LIN {X 0,Y 464.494,Z 1183.228,A -85,B 0,C 180,E1 15563.324,E2 15563.324} C_VEL
LIN {X 0,Y 465.219,Z 1176.701,A -85,B 0,C 180,E1 15560.224,E2 15560.224} C_VEL
LIN {X 0,Y 466.194,Z 1170.108,A -85,B 0,C 180,E1 15557.615,E2 15557.615} C_VEL
LIN {X 0,Y 467.574,Z 1162.416,A -85,B 0,C 180,E1 15555.004,E2 15555.004} C_VEL
LIN {X 0,Y 469.489,Z 1153.124,A -85,B 0,C 180,E1 15552.269,E2 15552.269} C_VEL
LIN {X 0,Y 472.708,Z 1139.667,A -85,B 0,C 180,E1 15548.88,E2 15548.88} C_VEL
LIN {X 0,Y 475.924,Z 1127.311,A -85,B 0,C 180,E1 15546.21,E2 15546.21} C_VEL
LIN {X 0,Y 479.291,Z 1115.185,A -85,B 0,C 180,E1 15543.884,E2 15543.884} C_VEL
LIN {X 0,Y 482.99,Z 1102.43,A -85,B 0,C 180,E1 15541.701,E2 15541.701} C_VEL
LIN {X 0,Y 487.449,Z 1087.469,A -85,B 0,C 180,E1 15539.422,E2 15539.422} C_VEL
LIN {X 0,Y 493.552,Z 1066.908,A -85,B 0,C 180,E1 15536.7,E2 15536.7} C_VEL
LIN {X 0,Y 498.429,Z 1050.219,A -85,B 0,C 180,E1 15534.778,E2 15534.778} C_VEL
LIN {X 0,Y 503.252,Z 1033.414,A -85,B 0,C 180,E1 15533.057,E2 15533.057} C_VEL
LIN {X 0,Y 508.073,Z 1016.053,A -85,B 0,C 180,E1 15531.474,E2 15531.474} C_VEL
LIN {X 0,Y 513.784,Z 994.616,A -85,B 0,C 180,E1 15529.751,E2 15529.751} C_VEL
LIN {X 0,Y 519.62,Z 970.597,A -85,B 0,C 180,E1 15528.109,E2 15528.109} C_VEL
LIN {X 0,Y 524.036,Z 951.032,A -85,B 0,C 180,E1 15526.953,E2 15526.953} C_VEL
LIN {X 0,Y 527.937,Z 932.043,A -85,B 0,C 180,E1 15525.967,E2 15525.967} C_VEL
LIN {X 0,Y 531.669,Z 912.17,A -85,B 0,C 180,E1 15525.075,E2 15525.075} C_VEL
LIN {X 0,Y 535.289,Z 890.47,A -85,B 0,C 180,E1 15524.246,E2 15524.246} C_VEL
LIN {X 0,Y 539.188,Z 862.655,A -85,B 0,C 180,E1 15523.385,E2 15523.385} C_VEL
LIN {X 0,Y 541.832,Z 838.413,A -85,B 0,C 180,E1 15522.811,E2 15522.811} C_VEL
LIN {X 0,Y 543.64,Z 816.068,A -85,B 0,C 180,E1 15522.403,E2 15522.403} C_VEL
LIN {X 0,Y 553.541,Z 604.138,A -85,B 0,C 180,E1 15519.202,E2 15519.202} C_VEL
LIN {X 0,Y 559.827,Z 471.624,A -85,B 0,C 180,E1 15517.173,E2 15517.173} C_VEL
LIN {X 0,Y 549.211,Z 455.582,A -85,B 0,C 180,E1 15515.058,E2 15515.058} C_VEL
LIN {X 0,Y 537.64,Z 439.734,A -85,B 0,C 180,E1 15512.544,E2 15512.544} C_VEL
LIN {X 0,Y 528.377,Z 427.759,A -85,B 0,C 180,E1 15510.318,E2 15510.318} C_VEL
LIN {X 0,Y 521.179,Z 418.584,A -85,B 0,C 180,E1 15508.411,E2 15508.411} C_VEL
LIN {X 0,Y 516.1,Z 412.456,A -85,B 0,C 180,E1 15506.959,E2 15506.959} C_VEL
LIN {X 0,Y 511.821,Z 407.184,A -85,B 0,C 180,E1 15505.641,E2 15505.641} C_VEL
LIN {X 0,Y 508.019,Z 402.462,A -85,B 0,C 180,E1 15504.383,E2 15504.383} C_VEL
LIN {X 0,Y 503.556,Z 397.56,A -85,B 0,C 180,E1 15502.812,E2 15502.812} C_VEL
LIN {X 0,Y 502.199,Z 395.757,A -85,B 0,C 180,E1 15502.29,E2 15502.29} C_VEL
LIN {X 0,Y 498.68,Z 392.223,A -85,B 0,C 180,E1 15500.91,E2 15500.91} C_VEL
LIN {X 0,Y 496.917,Z 389.555,A -85,B 0,C 180,E1 15500.126,E2 15500.126} C_VEL
LIN {X 0,Y 493.635,Z 386.766,A -85,B 0,C 180,E1 15498.665,E2 15498.665} C_VEL
LIN {X 0,Y 491.477,Z 383.313,A -85,B 0,C 180,E1 15497.524,E2 15497.524} C_VEL
LIN {X 0,Y 488.072,Z 380.844,A -85,B 0,C 180,E1 15495.69,E2 15495.69} C_VEL
LIN {X 0,Y 486.117,Z 377.519,A -85,B 0,C 180,E1 15494.353,E2 15494.353} C_VEL
LIN {X 0,Y 485.736,Z 376.677,A -85,B 0,C 180,E1 15494.058,E2 15494.058} C_VEL
LIN {X 0,Y 481.79,Z 374.262,A -85,B 0,C 180,E1 15490.997,E2 15490.997} C_VEL
LIN {X 0,Y 480.013,Z 370.955,A -85,B 0,C 180,E1 15488.807,E2 15488.807} C_VEL
LIN {X 0,Y 479.704,Z 369.991,A -85,B 0,C 180,E1 15488.269,E2 15488.269} C_VEL
LIN {X 0,Y 477.971,Z 369.512,A -85,B 0,C 180,E1 15481.558,E2 15481.558} C_VEL
LIN {X 0,Y 479.808,Z 370.162,A -85,B 0,C 180,E1 15477.671,E2 15477.671} C_VEL
LIN {X 0,Y 481.494,Z 373.959,A -85,B 0,C 180,E1 15475.4,E2 15475.4} C_VEL
LIN {X 0,Y 484.978,Z 376.507,A -85,B 0,C 180,E1 15472.537,E2 15472.537} C_VEL
LIN {X 0,Y 485.888,Z 377.026,A -85,B 0,C 180,E1 15471.926,E2 15471.926} C_VEL
LIN {X 0,Y 487.83,Z 380.574,A -85,B 0,C 180,E1 15470.562,E2 15470.562} C_VEL
LIN {X 0,Y 490.711,Z 382.963,A -85,B 0,C 180,E1 15468.957,E2 15468.957} C_VEL
LIN {X 0,Y 491.78,Z 383.73,A -85,B 0,C 180,E1 15468.417,E2 15468.417} C_VEL
LIN {X 0,Y 494.132,Z 387.367,A -85,B 0,C 180,E1 15467.198,E2 15467.198} C_VEL
LIN {X 0,Y 497.51,Z 390.286,A -85,B 0,C 180,E1 15465.718,E2 15465.718} C_VEL
LIN {X 0,Y 500.44,Z 394.393,A -85,B 0,C 180,E1 15464.47,E2 15464.47} C_VEL
LIN {X 0,Y 502.915,Z 396.596,A -85,B 0,C 180,E1 15463.542,E2 15463.542} C_VEL
LIN {X 0,Y 506.304,Z 400.928,A -85,B 0,C 180,E1 15462.294,E2 15462.294} C_VEL
LIN {X 0,Y 508.201,Z 402.882,A -85,B 0,C 180,E1 15461.651,E2 15461.651} C_VEL
LIN {X 0,Y 512.093,Z 407.534,A -85,B 0,C 180,E1 15460.376,E2 15460.376} C_VEL
LIN {X 0,Y 517.261,Z 413.691,A -85,B 0,C 180,E1 15458.809,E2 15458.809} C_VEL
LIN {X 0,Y 525.953,Z 424.62,A -85,B 0,C 180,E1 15456.41,E2 15456.41} C_VEL
LIN {X 0,Y 535.695,Z 438.163,A -85,B 0,C 180,E1 15453.983,E2 15453.983} C_VEL
LIN {X 0,Y 545.364,Z 452.379,A -85,B 0,C 180,E1 15451.799,E2 15451.799} C_VEL
LIN {X 0,Y 557.011,Z 470.151,A -85,B 0,C 180,E1 15449.409,E2 15449.409} C_VEL
LIN {X 0,Y 559.909,Z 475.043,A -85,B 0,C 180,E1 15448.84,E2 15448.84} C_VEL
LIN {X 0,Y 549.743,Z 688.806,A -85,B 0,C 180,E1 15445.603,E2 15445.603} C_VEL
LIN {X 0,Y 543.343,Z 825.734,A -85,B 0,C 180,E1 15443.532,E2 15443.532} C_VEL
LIN {X 0,Y 541.068,Z 852.241,A -85,B 0,C 180,E1 15443.031,E2 15443.031} C_VEL
LIN {X 0,Y 537.738,Z 879.381,A -85,B 0,C 180,E1 15442.329,E2 15442.329} C_VEL
LIN {X 0,Y 534.603,Z 900.655,A -85,B 0,C 180,E1 15441.641,E2 15441.641} C_VEL
LIN {X 0,Y 531.164,Z 921.015,A -85,B 0,C 180,E1 15440.856,E2 15440.856} C_VEL
LIN {X 0,Y 527.26,Z 941.653,A -85,B 0,C 180,E1 15439.924,E2 15439.924} C_VEL
LIN {X 0,Y 522.201,Z 965.926,A -85,B 0,C 180,E1 15438.641,E2 15438.641} C_VEL
LIN {X 0,Y 516.501,Z 990.068,A -85,B 0,C 180,E1 15437.116,E2 15437.116} C_VEL
LIN {X 0,Y 511.723,Z 1009.058,A -85,B 0,C 180,E1 15435.735,E2 15435.735} C_VEL
LIN {X 0,Y 507.046,Z 1026.704,A -85,B 0,C 180,E1 15434.288,E2 15434.288} C_VEL
LIN {X 0,Y 502.23,Z 1044.16,A -85,B 0,C 180,E1 15432.68,E2 15432.68} C_VEL
LIN {X 0,Y 496.37,Z 1064.899,A -85,B 0,C 180,E1 15430.515,E2 15430.515} C_VEL
LIN {X 0,Y 490.599,Z 1084.424,A -85,B 0,C 180,E1 15428.137,E2 15428.137} C_VEL
LIN {X 0,Y 486.228,Z 1099.357,A -85,B 0,C 180,E1 15426.082,E2 15426.082} C_VEL
LIN {X 0,Y 482.148,Z 1113.462,A -85,B 0,C 180,E1 15423.908,E2 15423.908} C_VEL
LIN {X 0,Y 477.734,Z 1129.428,A -85,B 0,C 180,E1 15421.126,E2 15421.126} C_VEL
LIN {X 0,Y 473.845,Z 1143.812,A -85,B 0,C 180,E1 15418.208,E2 15418.208} C_VEL
LIN {X 0,Y 471.148,Z 1154.885,A -85,B 0,C 180,E1 15415.654,E2 15415.654} C_VEL
LIN {X 0,Y 468.98,Z 1164.684,A -85,B 0,C 180,E1 15413.098,E2 15413.098} C_VEL
LIN {X 0,Y 467.14,Z 1174.105,A -85,B 0,C 180,E1 15410.289,E2 15410.289} C_VEL
LIN {X 0,Y 465.524,Z 1184.102,A -85,B 0,C 180,E1 15406.727,E2 15406.727} C_VEL
LIN {X 0,Y 464.749,Z 1190.478,A -85,B 0,C 180,E1 15403.944,E2 15403.944} C_VEL
LIN {X 0,Y 464.276,Z 1195.451,A -85,B 0,C 180,E1 15401.302,E2 15401.302} C_VEL
LIN {X 0,Y 464.059,Z 1199.18,A -85,B 0,C 180,E1 15398.8,E2 15398.8} C_VEL
LIN {X 0,Y 463.954,Z 1201.955,A -85,B 0,C 180,E1 15396.311,E2 15396.311} C_VEL
LIN {X 0,Y 463.914,Z 1203.811,A -85,B 0,C 180,E1 15393.832,E2 15393.832} C_VEL
LIN {X 0,Y 463.913,Z 1204.757,A -85,B 0,C 180,E1 15391.359,E2 15391.359} C_VEL
LIN {X 0,Y 463.911,Z 1204.802,A -85,B 0,C 180,E1 15388.889,E2 15388.889} C_VEL
LIN {X 0,Y 463.914,Z 1203.947,A -85,B 0,C 180,E1 15386.417,E2 15386.417} C_VEL
LIN {X 0,Y 463.946,Z 1202.182,A -85,B 0,C 180,E1 15383.939,E2 15383.939} C_VEL
LIN {X 0,Y 464.044,Z 1199.499,A -85,B 0,C 180,E1 15381.45,E2 15381.45} C_VEL
LIN {X 0,Y 464.247,Z 1195.869,A -85,B 0,C 180,E1 15378.949,E2 15378.949} C_VEL
LIN {X 0,Y 464.693,Z 1190.991,A -85,B 0,C 180,E1 15376.309,E2 15376.309} C_VEL
LIN {X 0,Y 465.386,Z 1185.016,A -85,B 0,C 180,E1 15373.654,E2 15373.654} C_VEL
LIN {X 0,Y 466.671,Z 1176.834,A -85,B 0,C 180,E1 15370.604,E2 15370.604} C_VEL
LIN {X 0,Y 468.695,Z 1166.062,A -85,B 0,C 180,E1 15367.287,E2 15367.287} C_VEL
LIN {X 0,Y 470.9,Z 1155.91,A -85,B 0,C 180,E1 15364.602,E2 15364.602} C_VEL
LIN {X 0,Y 473.409,Z 1145.524,A -85,B 0,C 180,E1 15362.176,E2 15362.176} C_VEL
LIN {X 0,Y 476.605,Z 1133.251,A -85,B 0,C 180,E1 15359.63,E2 15359.63} C_VEL
LIN {X 0,Y 481.304,Z 1116.552,A -85,B 0,C 180,E1 15356.598,E2 15356.598} C_VEL
LIN {X 0,Y 485.897,Z 1100.668,A -85,B 0,C 180,E1 15354.094,E2 15354.094} C_VEL
LIN {X 0,Y 490.374,Z 1085.712,A -85,B 0,C 180,E1 15351.992,E2 15351.992} C_VEL
LIN {X 0,Y 495.396,Z 1069.065,A -85,B 0,C 180,E1 15349.904,E2 15349.904} C_VEL
LIN {X 0,Y 501.936,Z 1047.346,A -85,B 0,C 180,E1 15347.523,E2 15347.523} C_VEL
LIN {X 0,Y 507.492,Z 1028.11,A -85,B 0,C 180,E1 15345.698,E2 15345.698} C_VEL
LIN {X 0,Y 512.501,Z 1010.212,A -85,B 0,C 180,E1 15344.195,E2 15344.195} C_VEL
LIN {X 0,Y 517.446,Z 991.688,A -85,B 0,C 180,E1 15342.815,E2 15342.815} C_VEL
LIN {X 0,Y 522.751,Z 970.617,A -85,B 0,C 180,E1 15341.438,E2 15341.438} C_VEL
LIN {X 0,Y 528.911,Z 943.682,A -85,B 0,C 180,E1 15339.954,E2 15339.954} C_VEL
LIN {X 0,Y 533.17,Z 922.749,A -85,B 0,C 180,E1 15338.984,E2 15338.984} C_VEL
LIN {X 0,Y 536.971,Z 901.909,A -85,B 0,C 180,E1 15338.164,E2 15338.164} C_VEL
LIN {X 0,Y 540.349,Z 880.681,A -85,B 0,C 180,E1 15337.463,E2 15337.463} C_VEL
LIN {X 0,Y 543.499,Z 857.212,A -85,B 0,C 180,E1 15336.834,E2 15336.834} C_VEL
LIN {X 0,Y 546.436,Z 827.726,A -85,B 0,C 180,E1 15336.245,E2 15336.245} C_VEL
LIN {X 0,Y 550.006,Z 762.107,A -85,B 0,C 180,E1 15335.225,E2 15335.225} C_VEL
LIN {X 0,Y 561.772,Z 540.644,A -85,B 0,C 180,E1 15331.826,E2 15331.826} C_VEL
LIN {X 0,Y 565.295,Z 475.693,A -85,B 0,C 180,E1 15330.802,E2 15330.802} C_VEL
LIN {X 0,Y 555.436,Z 460.281,A -85,B 0,C 180,E1 15328.434,E2 15328.434} C_VEL
LIN {X 0,Y 546.712,Z 447.485,A -85,B 0,C 180,E1 15326.095,E2 15326.095} C_VEL
LIN {X 0,Y 538.293,Z 435.817,A -85,B 0,C 180,E1 15323.539,E2 15323.539} C_VEL
LIN {X 0,Y 532.177,Z 427.926,A -85,B 0,C 180,E1 15321.435,E2 15321.435} C_VEL
LIN {X 0,Y 528.362,Z 423.112,A -85,B 0,C 180,E1 15319.974,E2 15319.974} C_VEL
LIN {X 0,Y 524.105,Z 418.212,A -85,B 0,C 180,E1 15318.176,E2 15318.176} C_VEL
LIN {X 0,Y 523.09,Z 416.707,A -85,B 0,C 180,E1 15317.694,E2 15317.694} C_VEL
LIN {X 0,Y 519.485,Z 412.975,A -85,B 0,C 180,E1 15315.919,E2 15315.919} C_VEL
LIN {X 0,Y 518.096,Z 410.63,A -85,B 0,C 180,E1 15315.102,E2 15315.102} C_VEL
LIN {X 0,Y 514.846,Z 407.925,A -85,B 0,C 180,E1 15313.134,E2 15313.134} C_VEL
LIN {X 0,Y 512.79,Z 404.278,A -85,B 0,C 180,E1 15311.472,E2 15311.472} C_VEL
LIN {X 0,Y 508.967,Z 401.286,A -85,B 0,C 180,E1 15307.45,E2 15307.45} C_VEL
LIN {X 0,Y 507.804,Z 397.837,A -85,B 0,C 180,E1 15303.726,E2 15303.726} C_VEL
LIN {X 0,Y 507.844,Z 398.021,A -85,B 0,C 180,E1 15301.692,E2 15301.692} C_VEL
LIN {X 0,Y 511.002,Z 403.337,A -85,B 0,C 180,E1 15295.848,E2 15295.848} C_VEL
LIN {X 0,Y 513.027,Z 404.558,A -85,B 0,C 180,E1 15294.127,E2 15294.127} C_VEL
LIN {X 0,Y 515.047,Z 408.114,A -85,B 0,C 180,E1 15292.526,E2 15292.526} C_VEL
LIN {X 0,Y 518.407,Z 411.102,A -85,B 0,C 180,E1 15290.508,E2 15290.508} C_VEL
LIN {X 0,Y 521.28,Z 415.186,A -85,B 0,C 180,E1 15288.941,E2 15288.941} C_VEL
LIN {X 0,Y 523.694,Z 417.451,A -85,B 0,C 180,E1 15287.82,E2 15287.82} C_VEL
LIN {X 0,Y 527.329,Z 422.013,A -85,B 0,C 180,E1 15286.233,E2 15286.233} C_VEL
LIN {X 0,Y 528.768,Z 423.671,A -85,B 0,C 180,E1 15285.657,E2 15285.657} C_VEL
LIN {X 0,Y 532.626,Z 428.31,A -85,B 0,C 180,E1 15284.204,E2 15284.204} C_VEL
LIN {X 0,Y 538.46,Z 435.74,A -85,B 0,C 180,E1 15282.214,E2 15282.214} C_VEL
LIN {X 0,Y 543.158,Z 441.816,A -85,B 0,C 180,E1 15280.76,E2 15280.76} C_VEL
LIN {X 0,Y 549.693,Z 450.264,A -85,B 0,C 180,E1 15278.918,E2 15278.918} C_VEL
LIN {X 0,Y 558.021,Z 461.797,A -85,B 0,C 180,E1 15276.783,E2 15276.783} C_VEL
LIN {X 0,Y 565.399,Z 473.165,A -85,B 0,C 180,E1 15275.041,E2 15275.041} C_VEL
LIN {X 0,Y 553.504,Z 691.017,A -85,B 0,C 180,E1 15271.688,E2 15271.688} C_VEL
LIN {X 0,Y 546.723,Z 818.932,A -85,B 0,C 180,E1 15269.718,E2 15269.718} C_VEL
LIN {X 0,Y 544.254,Z 845.823,A -85,B 0,C 180,E1 15269.199,E2 15269.199} C_VEL
LIN {X 0,Y 540.729,Z 872.618,A -85,B 0,C 180,E1 15268.49,E2 15268.49} C_VEL
LIN {X 0,Y 537.396,Z 893.834,A -85,B 0,C 180,E1 15267.789,E2 15267.789} C_VEL
LIN {X 0,Y 533.742,Z 914.094,A -85,B 0,C 180,E1 15266.992,E2 15266.992} C_VEL
LIN {X 0,Y 529.418,Z 935.44,A -85,B 0,C 180,E1 15266.006,E2 15266.006} C_VEL
LIN {X 0,Y 523.674,Z 960.883,A -85,B 0,C 180,E1 15264.615,E2 15264.615} C_VEL
LIN {X 0,Y 517.941,Z 983.544,A -85,B 0,C 180,E1 15263.138,E2 15263.138} C_VEL
LIN {X 0,Y 513.006,Z 1001.947,A -85,B 0,C 180,E1 15261.763,E2 15261.763} C_VEL
LIN {X 0,Y 508.11,Z 1019.32,A -85,B 0,C 180,E1 15260.301,E2 15260.301} C_VEL
LIN {X 0,Y 502.95,Z 1036.972,A -85,B 0,C 180,E1 15258.631,E2 15258.631} C_VEL
LIN {X 0,Y 496.464,Z 1058.496,A -85,B 0,C 180,E1 15256.304,E2 15256.304} C_VEL
LIN {X 0,Y 491.099,Z 1075.885,A -85,B 0,C 180,E1 15254.131,E2 15254.131} C_VEL
LIN {X 0,Y 486.456,Z 1091.107,A -85,B 0,C 180,E1 15251.99,E2 15251.99} C_VEL
LIN {X 0,Y 481.891,Z 1106.438,A -85,B 0,C 180,E1 15249.567,E2 15249.567} C_VEL
LIN {X 0,Y 476.887,Z 1123.885,A -85,B 0,C 180,E1 15246.395,E2 15246.395} C_VEL
LIN {X 0,Y 474.67,Z 1132.224,A -85,B 0,C 180,E1 15244.701,E2 15244.701} C_VEL
LIN {X 0,Y 472.708,Z 1136.071,A -85,B 0,C 180,E1 15243.914,E2 15243.914} C_VEL
LIN {X 0,Y 464.304,Z 1146.226,A -85,B 0,C 180,E1 15241.876,E2 15241.876} C_VEL
LIN {X 0,Y 462.881,Z 1149.176,A -85,B 0,C 180,E1 15241.164,E2 15241.164} C_VEL
LIN {X 0,Y 460.123,Z 1161.166,A -85,B 0,C 180,E1 15237.712,E2 15237.712} C_VEL
LIN {X 0,Y 458.484,Z 1169.521,A -85,B 0,C 180,E1 15234.873,E2 15234.873} C_VEL
LIN {X 0,Y 457.412,Z 1176.202,A -85,B 0,C 180,E1 15232.22,E2 15232.22} C_VEL
LIN {X 0,Y 456.694,Z 1181.827,A -85,B 0,C 180,E1 15229.57,E2 15229.57} C_VEL
LIN {X 0,Y 456.236,Z 1186.816,A -85,B 0,C 180,E1 15226.684,E2 15226.684} C_VEL
LIN {X 0,Y 455.983,Z 1191.277,A -85,B 0,C 180,E1 15223.19,E2 15223.19} C_VEL
LIN {X 0,Y 455.919,Z 1193.632,A -85,B 0,C 180,E1 15220.232,E2 15220.232} C_VEL
LIN {X 0,Y 455.912,Z 1194.733,A -85,B 0,C 180,E1 15217.556,E2 15217.556} C_VEL
LIN {X 0,Y 455.902,Z 1194.832,A -85,B 0,C 180,E1 15214.906,E2 15214.906} C_VEL
LIN {X 0,Y 455.916,Z 1194.011,A -85,B 0,C 180,E1 15212.388,E2 15212.388} C_VEL
LIN {X 0,Y 455.957,Z 1192.189,A -85,B 0,C 180,E1 15209.748,E2 15209.748} C_VEL
LIN {X 0,Y 456.064,Z 1189.388,A -85,B 0,C 180,E1 15207.109,E2 15207.109} C_VEL
LIN {X 0,Y 456.314,Z 1185.599,A -85,B 0,C 180,E1 15204.467,E2 15204.467} C_VEL
LIN {X 0,Y 456.837,Z 1180.558,A -85,B 0,C 180,E1 15201.694,E2 15201.694} C_VEL
LIN {X 0,Y 457.94,Z 1172.88,A -85,B 0,C 180,E1 15198.284,E2 15198.284} C_VEL
LIN {X 0,Y 459.603,Z 1163.651,A -85,B 0,C 180,E1 15195.006,E2 15195.006} C_VEL
LIN {X 0,Y 461.467,Z 1154.919,A -85,B 0,C 180,E1 15192.341,E2 15192.341} C_VEL
LIN {X 0,Y 463.928,Z 1144.806,A -85,B 0,C 180,E1 15189.644,E2 15189.644} C_VEL
LIN {X 0,Y 467.707,Z 1130.975,A -85,B 0,C 180,E1 15186.436,E2 15186.436} C_VEL
LIN {X 0,Y 471.828,Z 1116.503,A -85,B 0,C 180,E1 15183.575,E2 15183.575} C_VEL
LIN {X 0,Y 475.879,Z 1103.089,A -85,B 0,C 180,E1 15181.239,E2 15181.239} C_VEL
LIN {X 0,Y 480.239,Z 1088.965,A -85,B 0,C 180,E1 15179.051,E2 15179.051} C_VEL
LIN {X 0,Y 485.98,Z 1070.6,A -85,B 0,C 180,E1 15176.537,E2 15176.537} C_VEL
LIN {X 0,Y 491.885,Z 1050.963,A -85,B 0,C 180,E1 15174.231,E2 15174.231} C_VEL
LIN {X 0,Y 496.857,Z 1034.259,A -85,B 0,C 180,E1 15172.5,E2 15172.5} C_VEL
LIN {X 0,Y 501.836,Z 1016.951,A -85,B 0,C 180,E1 15170.905,E2 15170.905} C_VEL
LIN {X 0,Y 506.934,Z 998.422,A -85,B 0,C 180,E1 15169.391,E2 15169.391} C_VEL
LIN {X 0,Y 513.143,Z 974.34,A -85,B 0,C 180,E1 15167.684,E2 15167.684} C_VEL
LIN {X 0,Y 518.178,Z 952.749,A -85,B 0,C 180,E1 15166.383,E2 15166.383} C_VEL
LIN {X 0,Y 522.297,Z 933.395,A -85,B 0,C 180,E1 15165.365,E2 15165.365} C_VEL
LIN {X 0,Y 526.131,Z 913.682,A -85,B 0,C 180,E1 15164.47,E2 15164.47} C_VEL
LIN {X 0,Y 529.731,Z 892.912,A -85,B 0,C 180,E1 15163.665,E2 15163.665} C_VEL
LIN {X 0,Y 533.099,Z 870.397,A -85,B 0,C 180,E1 15162.935,E2 15162.935} C_VEL
LIN {X 0,Y 536.552,Z 841.46,A -85,B 0,C 180,E1 15162.204,E2 15162.204} C_VEL
LIN {X 0,Y 538.587,Z 817.735,A -85,B 0,C 180,E1 15161.761,E2 15161.761} C_VEL
LIN {X 0,Y 548.244,Z 618.409,A -85,B 0,C 180,E1 15158.735,E2 15158.735} C_VEL
LIN {X 0,Y 555.289,Z 475.965,A -85,B 0,C 180,E1 15156.557,E2 15156.557} C_VEL
LIN {X 0,Y 545.319,Z 460.849,A -85,B 0,C 180,E1 15154.512,E2 15154.512} C_VEL
LIN {X 0,Y 534.465,Z 445.995,A -85,B 0,C 180,E1 15152.095,E2 15152.095} C_VEL
LIN {X 0,Y 525.847,Z 434.673,A -85,B 0,C 180,E1 15149.975,E2 15149.975} C_VEL
LIN {X 0,Y 518.374,Z 425.162,A -85,B 0,C 180,E1 15147.952,E2 15147.952} C_VEL
LIN {X 0,Y 514.097,Z 419.837,A -85,B 0,C 180,E1 15146.698,E2 15146.698} C_VEL
LIN {X 0,Y 509.87,Z 414.581,A -85,B 0,C 180,E1 15145.372,E2 15145.372} C_VEL
LIN {X 0,Y 505.248,Z 409.009,A -85,B 0,C 180,E1 15143.811,E2 15143.811} C_VEL
LIN {X 0,Y 501.515,Z 404.619,A -85,B 0,C 180,E1 15142.445,E2 15142.445} C_VEL
LIN {X 0,Y 500.229,Z 403.131,A -85,B 0,C 180,E1 15141.95,E2 15141.95} C_VEL
LIN {X 0,Y 496.677,Z 399.227,A -85,B 0,C 180,E1 15140.505,E2 15140.505} C_VEL
LIN {X 0,Y 495.446,Z 397.292,A -85,B 0,C 180,E1 15139.942,E2 15139.942} C_VEL
LIN {X 0,Y 492.093,Z 394.327,A -85,B 0,C 180,E1 15138.419,E2 15138.419} C_VEL
LIN {X 0,Y 490.072,Z 391.102,A -85,B 0,C 180,E1 15137.331,E2 15137.331} C_VEL
LIN {X 0,Y 486.545,Z 388.328,A -85,B 0,C 180,E1 15135.373,E2 15135.373} C_VEL
LIN {X 0,Y 484.661,Z 384.891,A -85,B 0,C 180,E1 15134.029,E2 15134.029} C_VEL
LIN {X 0,Y 480.258,Z 381.564,A -85,B 0,C 180,E1 15130.436,E2 15130.436} C_VEL
LIN {X 0,Y 478.819,Z 378.389,A -85,B 0,C 180,E1 15128.466,E2 15128.466} C_VEL
LIN {X 0,Y 478.563,Z 377.91,A -85,B 0,C 180,E1 15128.047,E2 15128.047} C_VEL
LIN {X 0,Y 476.994,Z 377.452,A -85,B 0,C 180,E1 15121.562,E2 15121.562} C_VEL
LIN {X 0,Y 478.738,Z 378.117,A -85,B 0,C 180,E1 15117.786,E2 15117.786} C_VEL
LIN {X 0,Y 480.465,Z 381.914,A -85,B 0,C 180,E1 15115.438,E2 15115.438} C_VEL
LIN {X 0,Y 484.008,Z 384.457,A -85,B 0,C 180,E1 15112.522,E2 15112.522} C_VEL
LIN {X 0,Y 484.673,Z 385.047,A -85,B 0,C 180,E1 15112.055,E2 15112.055} C_VEL
LIN {X 0,Y 486.935,Z 388.827,A -85,B 0,C 180,E1 15110.485,E2 15110.485} C_VEL
LIN {X 0,Y 490.348,Z 391.501,A -85,B 0,C 180,E1 15108.622,E2 15108.622} C_VEL
LIN {X 0,Y 492.912,Z 395.292,A -85,B 0,C 180,E1 15107.285,E2 15107.285} C_VEL
LIN {X 0,Y 495.937,Z 397.969,A -85,B 0,C 180,E1 15105.939,E2 15105.939} C_VEL
LIN {X 0,Y 499.043,Z 402.208,A -85,B 0,C 180,E1 15104.605,E2 15104.605} C_VEL
LIN {X 0,Y 501.268,Z 404.296,A -85,B 0,C 180,E1 15103.754,E2 15103.754} C_VEL
LIN {X 0,Y 504.865,Z 408.75,A -85,B 0,C 180,E1 15102.42,E2 15102.42} C_VEL
LIN {X 0,Y 506.495,Z 410.591,A -85,B 0,C 180,E1 15101.855,E2 15101.855} C_VEL
LIN {X 0,Y 511.423,Z 416.606,A -85,B 0,C 180,E1 15100.231,E2 15100.231} C_VEL
LIN {X 0,Y 516.602,Z 422.974,A -85,B 0,C 180,E1 15098.661,E2 15098.661} C_VEL
LIN {X 0,Y 521.526,Z 429.182,A -85,B 0,C 180,E1 15097.274,E2 15097.274} C_VEL
LIN {X 0,Y 527.941,Z 437.77,A -85,B 0,C 180,E1 15095.584,E2 15095.584} C_VEL
LIN {X 0,Y 539.173,Z 453.971,A -85,B 0,C 180,E1 15092.887,E2 15092.887} C_VEL
LIN {X 0,Y 552.285,Z 474.112,A -85,B 0,C 180,E1 15090.08,E2 15090.08} C_VEL
LIN {X 0,Y 555.305,Z 479.278,A -85,B 0,C 180,E1 15089.468,E2 15089.468} C_VEL
LIN {X 0,Y 544.831,Z 692.393,A -85,B 0,C 180,E1 15086.227,E2 15086.227} C_VEL
LIN {X 0,Y 538.38,Z 825.7,A -85,B 0,C 180,E1 15084.2,E2 15084.2} C_VEL
LIN {X 0,Y 536.018,Z 852.514,A -85,B 0,C 180,E1 15083.692,E2 15083.692} C_VEL
LIN {X 0,Y 532.612,Z 879.444,A -85,B 0,C 180,E1 15082.993,E2 15082.993} C_VEL
LIN {X 0,Y 529.417,Z 900.516,A -85,B 0,C 180,E1 15082.311,E2 15082.311} C_VEL
LIN {X 0,Y 525.881,Z 920.881,A -85,B 0,C 180,E1 15081.525,E2 15081.525} C_VEL
LIN {X 0,Y 521.995,Z 940.841,A -85,B 0,C 180,E1 15080.624,E2 15080.624} C_VEL
LIN {X 0,Y 517.349,Z 962.6,A -85,B 0,C 180,E1 15079.481,E2 15079.481} C_VEL
LIN {X 0,Y 511.266,Z 988.087,A -85,B 0,C 180,E1 15077.901,E2 15077.901} C_VEL
LIN {X 0,Y 506.133,Z 1007.868,A -85,B 0,C 180,E1 15076.471,E2 15076.471} C_VEL
LIN {X 0,Y 501.422,Z 1025.079,A -85,B 0,C 180,E1 15075.065,E2 15075.065} C_VEL
LIN {X 0,Y 496.431,Z 1042.571,A -85,B 0,C 180,E1 15073.459,E2 15073.459} C_VEL
LIN {X 0,Y 491.379,Z 1059.733,A -85,B 0,C 180,E1 15071.686,E2 15071.686} C_VEL
LIN {X 0,Y 485.197,Z 1080.426,A -85,B 0,C 180,E1 15069.247,E2 15069.247} C_VEL
LIN {X 0,Y 479.818,Z 1097.962,A -85,B 0,C 180,E1 15066.849,E2 15066.849} C_VEL
LIN {X 0,Y 475.626,Z 1111.821,A -85,B 0,C 180,E1 15064.716,E2 15064.716} C_VEL
LIN {X 0,Y 471.694,Z 1125.063,A -85,B 0,C 180,E1 15062.432,E2 15062.432} C_VEL
LIN {X 0,Y 467.801,Z 1138.941,A -85,B 0,C 180,E1 15059.728,E2 15059.728} C_VEL
LIN {X 0,Y 463.994,Z 1153.235,A -85,B 0,C 180,E1 15056.492,E2 15056.492} C_VEL
LIN {X 0,Y 461.509,Z 1163.667,A -85,B 0,C 180,E1 15053.765,E2 15053.765} C_VEL
LIN {X 0,Y 459.668,Z 1172.38,A -85,B 0,C 180,E1 15051.167,E2 15051.167} C_VEL
LIN {X 0,Y 458.279,Z 1179.958,A -85,B 0,C 180,E1 15048.575,E2 15048.575} C_VEL
LIN {X 0,Y 457.184,Z 1187.375,A -85,B 0,C 180,E1 15045.606,E2 15045.606} C_VEL
LIN {X 0,Y 456.407,Z 1194.319,A -85,B 0,C 180,E1 15042.141,E2 15042.141} C_VEL
LIN {X 0,Y 456.083,Z 1198.787,A -85,B 0,C 180,E1 15039.21,E2 15039.21} C_VEL
LIN {X 0,Y 455.961,Z 1201.797,A -85,B 0,C 180,E1 15036.548,E2 15036.548} C_VEL
LIN {X 0,Y 455.915,Z 1203.718,A -85,B 0,C 180,E1 15034.025,E2 15034.025} C_VEL
LIN {X 0,Y 455.91,Z 1204.722,A -85,B 0,C 180,E1 15031.509,E2 15031.509} C_VEL
LIN {X 0,Y 455.908,Z 1204.814,A -85,B 0,C 180,E1 15028.995,E2 15028.995} C_VEL
LIN {X 0,Y 455.914,Z 1203.993,A -85,B 0,C 180,E1 15026.48,E2 15026.48} C_VEL
LIN {X 0,Y 455.946,Z 1202.256,A -85,B 0,C 180,E1 15023.958,E2 15023.958} C_VEL
LIN {X 0,Y 456.046,Z 1199.593,A -85,B 0,C 180,E1 15021.426,E2 15021.426} C_VEL
LIN {X 0,Y 456.256,Z 1195.986,A -85,B 0,C 180,E1 15018.881,E2 15018.881} C_VEL
LIN {X 0,Y 456.723,Z 1191.155,A -85,B 0,C 180,E1 15016.195,E2 15016.195} C_VEL
LIN {X 0,Y 457.405,Z 1185.533,A -85,B 0,C 180,E1 15013.622,E2 15013.622} C_VEL
LIN {X 0,Y 458.53,Z 1178.521,A -85,B 0,C 180,E1 15010.908,E2 15010.908} C_VEL
LIN {X 0,Y 460.416,Z 1168.771,A -85,B 0,C 180,E1 15007.691,E2 15007.691} C_VEL
LIN {X 0,Y 463.098,Z 1156.847,A -85,B 0,C 180,E1 15004.417,E2 15004.417} C_VEL
LIN {X 0,Y 465.835,Z 1145.999,A -85,B 0,C 180,E1 15001.823,E2 15001.823} C_VEL
LIN {X 0,Y 469.183,Z 1133.802,A -85,B 0,C 180,E1 14999.239,E2 14999.239} C_VEL
LIN {X 0,Y 473.868,Z 1118.065,A -85,B 0,C 180,E1 14996.294,E2 14996.294} C_VEL
LIN {X 0,Y 479.13,Z 1100.698,A -85,B 0,C 180,E1 14993.506,E2 14993.506} C_VEL
LIN {X 0,Y 483.844,Z 1085.67,A -85,B 0,C 180,E1 14991.367,E2 14991.367} C_VEL
LIN {X 0,Y 489.017,Z 1069.294,A -85,B 0,C 180,E1 14989.289,E2 14989.289} C_VEL
LIN {X 0,Y 495.696,Z 1048.068,A -85,B 0,C 180,E1 14986.931,E2 14986.931} C_VEL
LIN {X 0,Y 501.818,Z 1027.675,A -85,B 0,C 180,E1 14984.982,E2 14984.982} C_VEL
LIN {X 0,Y 506.915,Z 1010.153,A -85,B 0,C 180,E1 14983.504,E2 14983.504} C_VEL
LIN {X 0,Y 511.885,Z 992.218,A -85,B 0,C 180,E1 14982.16,E2 14982.16} C_VEL
LIN {X 0,Y 517.138,Z 972.061,A -85,B 0,C 180,E1 14980.831,E2 14980.831} C_VEL
LIN {X 0,Y 523.305,Z 946.433,A -85,B 0,C 180,E1 14979.388,E2 14979.388} C_VEL
LIN {X 0,Y 528.165,Z 923.368,A -85,B 0,C 180,E1 14978.308,E2 14978.308} C_VEL
LIN {X 0,Y 532.074,Z 902.633,A -85,B 0,C 180,E1 14977.488,E2 14977.488} C_VEL
LIN {X 0,Y 535.588,Z 881.307,A -85,B 0,C 180,E1 14976.78,E2 14976.78} C_VEL
LIN {X 0,Y 538.665,Z 859.205,A -85,B 0,C 180,E1 14976.181,E2 14976.181} C_VEL
LIN {X 0,Y 541.716,Z 831.12,A -85,B 0,C 180,E1 14975.6,E2 14975.6} C_VEL
LIN {X 0,Y 544.495,Z 783.901,A -85,B 0,C 180,E1 14974.852,E2 14974.852} C_VEL
LIN {X 0,Y 556.677,Z 560.881,A -85,B 0,C 180,E1 14971.421,E2 14971.421} C_VEL
LIN {X 0,Y 561.25,Z 480.305,A -85,B 0,C 180,E1 14970.159,E2 14970.159} C_VEL
LIN {X 0,Y 552.129,Z 466.017,A -85,B 0,C 180,E1 14967.896,E2 14967.896} C_VEL
LIN {X 0,Y 544.433,Z 454.541,A -85,B 0,C 180,E1 14965.773,E2 14965.773} C_VEL
LIN {X 0,Y 536.232,Z 442.992,A -85,B 0,C 180,E1 14963.227,E2 14963.227} C_VEL
LIN {X 0,Y 530.36,Z 435.348,A -85,B 0,C 180,E1 14961.164,E2 14961.164} C_VEL
LIN {X 0,Y 525.958,Z 429.862,A -85,B 0,C 180,E1 14959.432,E2 14959.432} C_VEL
LIN {X 0,Y 522.442,Z 425.591,A -85,B 0,C 180,E1 14957.889,E2 14957.889} C_VEL
LIN {X 0,Y 521.43,Z 424.254,A -85,B 0,C 180,E1 14957.406,E2 14957.406} C_VEL
LIN {X 0,Y 517.832,Z 420.239,A -85,B 0,C 180,E1 14955.569,E2 14955.569} C_VEL
LIN {X 0,Y 516.544,Z 418.306,A -85,B 0,C 180,E1 14954.804,E2 14954.804} C_VEL
LIN {X 0,Y 513.413,Z 415.414,A -85,B 0,C 180,E1 14952.828,E2 14952.828} C_VEL
LIN {X 0,Y 511.685,Z 412.18,A -85,B 0,C 180,E1 14951.383,E2 14951.383} C_VEL
LIN {X 0,Y 507.925,Z 409.17,A -85,B 0,C 180,E1 14947.352,E2 14947.352} C_VEL
LIN {X 0,Y 506.828,Z 405.778,A -85,B 0,C 180,E1 14943.733,E2 14943.733} C_VEL
LIN {X 0,Y 506.859,Z 406.018,A -85,B 0,C 180,E1 14941.696,E2 14941.696} C_VEL
LIN {X 0,Y 510.025,Z 411.298,A -85,B 0,C 180,E1 14935.84,E2 14935.84} C_VEL
LIN {X 0,Y 511.894,Z 412.55,A -85,B 0,C 180,E1 14934.226,E2 14934.226} C_VEL
LIN {X 0,Y 514.062,Z 416.181,A -85,B 0,C 180,E1 14932.512,E2 14932.512} C_VEL
LIN {X 0,Y 517.037,Z 418.805,A -85,B 0,C 180,E1 14930.707,E2 14930.707} C_VEL
LIN {X 0,Y 519.971,Z 422.976,A -85,B 0,C 180,E1 14929.081,E2 14929.081} C_VEL
LIN {X 0,Y 522.237,Z 425.165,A -85,B 0,C 180,E1 14928.01,E2 14928.01} C_VEL
LIN {X 0,Y 525.959,Z 429.806,A -85,B 0,C 180,E1 14926.365,E2 14926.365} C_VEL
LIN {X 0,Y 527.625,Z 431.984,A -85,B 0,C 180,E1 14925.682,E2 14925.682} C_VEL
LIN {X 0,Y 532.039,Z 437.427,A -85,B 0,C 180,E1 14924.018,E2 14924.018} C_VEL
LIN {X 0,Y 536.6,Z 443.188,A -85,B 0,C 180,E1 14922.458,E2 14922.458} C_VEL
LIN {X 0,Y 541.569,Z 449.697,A -85,B 0,C 180,E1 14920.898,E2 14920.898} C_VEL
LIN {X 0,Y 548.133,Z 458.42,A -85,B 0,C 180,E1 14919.023,E2 14919.023} C_VEL
LIN {X 0,Y 555.741,Z 469.051,A -85,B 0,C 180,E1 14917.047,E2 14917.047} C_VEL
LIN {X 0,Y 561.32,Z 477.852,A -85,B 0,C 180,E1 14915.689,E2 14915.689} C_VEL
LIN {X 0,Y 549.099,Z 694.408,A -85,B 0,C 180,E1 14912.347,E2 14912.347} C_VEL
LIN {X 0,Y 542.256,Z 819.068,A -85,B 0,C 180,E1 14910.419,E2 14910.419} C_VEL
LIN {X 0,Y 539.698,Z 846.12,A -85,B 0,C 180,E1 14909.897,E2 14909.897} C_VEL
LIN {X 0,Y 536.087,Z 872.741,A -85,B 0,C 180,E1 14909.192,E2 14909.192} C_VEL
LIN {X 0,Y 532.703,Z 893.662,A -85,B 0,C 180,E1 14908.502,E2 14908.502} C_VEL
LIN {X 0,Y 528.979,Z 913.765,A -85,B 0,C 180,E1 14907.713,E2 14907.713} C_VEL
LIN {X 0,Y 524.723,Z 934.195,A -85,B 0,C 180,E1 14906.774,E2 14906.774} C_VEL
LIN {X 0,Y 519.606,Z 956.527,A -85,B 0,C 180,E1 14905.573,E2 14905.573} C_VEL
LIN {X 0,Y 513.114,Z 981.72,A -85,B 0,C 180,E1 14903.967,E2 14903.967} C_VEL
LIN {X 0,Y 507.948,Z 1000.358,A -85,B 0,C 180,E1 14902.586,E2 14902.586} C_VEL
LIN {X 0,Y 502.834,Z 1017.864,A -85,B 0,C 180,E1 14901.122,E2 14901.122} C_VEL
LIN {X 0,Y 497.433,Z 1035.631,A -85,B 0,C 180,E1 14899.446,E2 14899.446} C_VEL
LIN {X 0,Y 491.313,Z 1055.343,A -85,B 0,C 180,E1 14897.335,E2 14897.335} C_VEL
LIN {X 0,Y 484.861,Z 1075.319,A -85,B 0,C 180,E1 14894.85,E2 14894.85} C_VEL
LIN {X 0,Y 480.123,Z 1090.118,A -85,B 0,C 180,E1 14892.758,E2 14892.758} C_VEL
LIN {X 0,Y 475.629,Z 1104.323,A -85,B 0,C 180,E1 14890.51,E2 14890.51} C_VEL
LIN {X 0,Y 471.097,Z 1119.317,A -85,B 0,C 180,E1 14887.834,E2 14887.834} C_VEL
LIN {X 0,Y 466.608,Z 1134.825,A -85,B 0,C 180,E1 14884.626,E2 14884.626} C_VEL
LIN {X 0,Y 463.706,Z 1145.75,A -85,B 0,C 180,E1 14882.035,E2 14882.035} C_VEL
LIN {X 0,Y 462.881,Z 1149.176,A -85,B 0,C 180,E1 14881.164,E2 14881.164} C_VEL
LIN {X 0,Y 461.14,Z 1152.549,A -85,B 0,C 180,E1 14880.324,E2 14880.324} C_VEL
LIN {X 0,Y 453.162,Z 1161.156,A -85,B 0,C 180,E1 14878.099,E2 14878.099} C_VEL
LIN {X 0,Y 451.898,Z 1163.599,A -85,B 0,C 180,E1 14877.332,E2 14877.332} C_VEL
LIN {X 0,Y 450.215,Z 1172.147,A -85,B 0,C 180,E1 14874.258,E2 14874.258} C_VEL
LIN {X 0,Y 448.972,Z 1180.193,A -85,B 0,C 180,E1 14870.712,E2 14870.712} C_VEL
LIN {X 0,Y 448.38,Z 1185.482,A -85,B 0,C 180,E1 14867.783,E2 14867.783} C_VEL
LIN {X 0,Y 448.091,Z 1189.266,A -85,B 0,C 180,E1 14865.133,E2 14865.133} C_VEL
LIN {X 0,Y 447.959,Z 1192.076,A -85,B 0,C 180,E1 14862.504,E2 14862.504} C_VEL
LIN {X 0,Y 447.916,Z 1193.936,A -85,B 0,C 180,E1 14859.897,E2 14859.897} C_VEL
LIN {X 0,Y 447.915,Z 1194.869,A -85,B 0,C 180,E1 14857.31,E2 14857.31} C_VEL
LIN {X 0,Y 447.903,Z 1194.893,A -85,B 0,C 180,E1 14854.737,E2 14854.737} C_VEL
LIN {X 0,Y 447.92,Z 1194.02,A -85,B 0,C 180,E1 14852.174,E2 14852.174} C_VEL
LIN {X 0,Y 447.962,Z 1192.258,A -85,B 0,C 180,E1 14849.616,E2 14849.616} C_VEL
LIN {X 0,Y 448.082,Z 1189.45,A -85,B 0,C 180,E1 14846.93,E2 14846.93} C_VEL
LIN {X 0,Y 448.359,Z 1185.655,A -85,B 0,C 180,E1 14844.24,E2 14844.24} C_VEL
LIN {X 0,Y 448.91,Z 1180.606,A -85,B 0,C 180,E1 14841.417,E2 14841.417} C_VEL
LIN {X 0,Y 450.104,Z 1172.917,A -85,B 0,C 180,E1 14837.947,E2 14837.947} C_VEL
LIN {X 0,Y 451.805,Z 1164.042,A -85,B 0,C 180,E1 14834.73,E2 14834.73} C_VEL
LIN {X 0,Y 453.862,Z 1154.941,A -85,B 0,C 180,E1 14831.902,E2 14831.902} C_VEL
LIN {X 0,Y 456.41,Z 1145.019,A -85,B 0,C 180,E1 14829.212,E2 14829.212} C_VEL
LIN {X 0,Y 460.11,Z 1132.134,A -85,B 0,C 180,E1 14826.158,E2 14826.158} C_VEL
LIN {X 0,Y 464.579,Z 1117.107,A -85,B 0,C 180,E1 14823.13,E2 14823.13} C_VEL
LIN {X 0,Y 468.796,Z 1103.715,A -85,B 0,C 180,E1 14820.762,E2 14820.762} C_VEL
LIN {X 0,Y 473.312,Z 1089.62,A -85,B 0,C 180,E1 14818.547,E2 14818.547} C_VEL
LIN {X 0,Y 478.954,Z 1072.194,A -85,B 0,C 180,E1 14816.124,E2 14816.124} C_VEL
LIN {X 0,Y 485.193,Z 1052.331,A -85,B 0,C 180,E1 14813.74,E2 14813.74} C_VEL
LIN {X 0,Y 490.679,Z 1034.496,A -85,B 0,C 180,E1 14811.871,E2 14811.871} C_VEL
LIN {X 0,Y 495.833,Z 1017.184,A -85,B 0,C 180,E1 14810.264,E2 14810.264} C_VEL
LIN {X 0,Y 501.096,Z 998.675,A -85,B 0,C 180,E1 14808.742,E2 14808.742} C_VEL
LIN {X 0,Y 507.505,Z 974.576,A -85,B 0,C 180,E1 14807.024,E2 14807.024} C_VEL
LIN {X 0,Y 512.809,Z 952.499,A -85,B 0,C 180,E1 14805.692,E2 14805.692} C_VEL
LIN {X 0,Y 517.168,Z 932.547,A -85,B 0,C 180,E1 14804.644,E2 14804.644} C_VEL
LIN {X 0,Y 521.125,Z 912.684,A -85,B 0,C 180,E1 14803.748,E2 14803.748} C_VEL
LIN {X 0,Y 524.824,Z 891.725,A -85,B 0,C 180,E1 14802.94,E2 14802.94} C_VEL
LIN {X 0,Y 528.864,Z 865.058,A -85,B 0,C 180,E1 14802.097,E2 14802.097} C_VEL
LIN {X 0,Y 531.858,Z 839.126,A -85,B 0,C 180,E1 14801.476,E2 14801.476} C_VEL
LIN {X 0,Y 533.788,Z 816.61,A -85,B 0,C 180,E1 14801.061,E2 14801.061} C_VEL
LIN {X 0,Y 544.344,Z 605.533,A -85,B 0,C 180,E1 14797.844,E2 14797.844} C_VEL
LIN {X 0,Y 550.687,Z 480.242,A -85,B 0,C 180,E1 14795.908,E2 14795.908} C_VEL
LIN {X 0,Y 542.239,Z 467.309,A -85,B 0,C 180,E1 14794.128,E2 14794.128} C_VEL
LIN {X 0,Y 531.737,Z 452.767,A -85,B 0,C 180,E1 14791.739,E2 14791.739} C_VEL
LIN {X 0,Y 523.153,Z 441.343,A -85,B 0,C 180,E1 14789.58,E2 14789.58} C_VEL
LIN {X 0,Y 515.967,Z 432.126,A -85,B 0,C 180,E1 14787.591,E2 14787.591} C_VEL
LIN {X 0,Y 511.757,Z 426.836,A -85,B 0,C 180,E1 14786.329,E2 14786.329} C_VEL
LIN {X 0,Y 507.764,Z 421.807,A -85,B 0,C 180,E1 14785.048,E2 14785.048} C_VEL
LIN {X 0,Y 503.369,Z 416.434,A -85,B 0,C 180,E1 14783.532,E2 14783.532} C_VEL
LIN {X 0,Y 499.562,Z 411.784,A -85,B 0,C 180,E1 14782.104,E2 14782.104} C_VEL
LIN {X 0,Y 494.946,Z 406.607,A -85,B 0,C 180,E1 14780.21,E2 14780.21} C_VEL
LIN {X 0,Y 493.718,Z 404.859,A -85,B 0,C 180,E1 14779.645,E2 14779.645} C_VEL
LIN {X 0,Y 490.34,Z 401.582,A -85,B 0,C 180,E1 14778.057,E2 14778.057} C_VEL
LIN {X 0,Y 488.674,Z 398.883,A -85,B 0,C 180,E1 14777.136,E2 14777.136} C_VEL
LIN {X 0,Y 485.123,Z 395.916,A -85,B 0,C 180,E1 14775.113,E2 14775.113} C_VEL
LIN {X 0,Y 483.12,Z 392.368,A -85,B 0,C 180,E1 14773.647,E2 14773.647} C_VEL
LIN {X 0,Y 479.396,Z 389.758,A -85,B 0,C 180,E1 14770.576,E2 14770.576} C_VEL
LIN {X 0,Y 477.757,Z 386.356,A -85,B 0,C 180,E1 14768.364,E2 14768.364} C_VEL
LIN {X 0,Y 477.49,Z 385.836,A -85,B 0,C 180,E1 14767.913,E2 14767.913} C_VEL
LIN {X 0,Y 476.042,Z 385.403,A -85,B 0,C 180,E1 14761.444,E2 14761.444} C_VEL
LIN {X 0,Y 477.673,Z 386.051,A -85,B 0,C 180,E1 14757.901,E2 14757.901} C_VEL
LIN {X 0,Y 479.458,Z 389.894,A -85,B 0,C 180,E1 14755.455,E2 14755.455} C_VEL
LIN {X 0,Y 483.038,Z 392.407,A -85,B 0,C 180,E1 14752.507,E2 14752.507} C_VEL
LIN {X 0,Y 483.8,Z 393.768,A -85,B 0,C 180,E1 14751.921,E2 14751.921} C_VEL
LIN {X 0,Y 486.635,Z 397.583,A -85,B 0,C 180,E1 14750.061,E2 14750.061} C_VEL
LIN {X 0,Y 488.974,Z 399.348,A -85,B 0,C 180,E1 14748.798,E2 14748.798} C_VEL
LIN {X 0,Y 491.694,Z 403.21,A -85,B 0,C 180,E1 14747.373,E2 14747.373} C_VEL
LIN {X 0,Y 494.373,Z 405.638,A -85,B 0,C 180,E1 14746.163,E2 14746.163} C_VEL
LIN {X 0,Y 497.65,Z 410.019,A -85,B 0,C 180,E1 14744.739,E2 14744.739} C_VEL
LIN {X 0,Y 499.631,Z 411.977,A -85,B 0,C 180,E1 14743.968,E2 14743.968} C_VEL
LIN {X 0,Y 503.428,Z 416.568,A -85,B 0,C 180,E1 14742.548,E2 14742.548} C_VEL
LIN {X 0,Y 509.512,Z 424.08,A -85,B 0,C 180,E1 14740.482,E2 14740.482} C_VEL
LIN {X 0,Y 514.807,Z 430.68,A -85,B 0,C 180,E1 14738.852,E2 14738.852} C_VEL
LIN {X 0,Y 521.185,Z 438.724,A -85,B 0,C 180,E1 14737.052,E2 14737.052} C_VEL
LIN {X 0,Y 530.592,Z 452.201,A -85,B 0,C 180,E1 14734.614,E2 14734.614} C_VEL
LIN {X 0,Y 539.618,Z 465.792,A -85,B 0,C 180,E1 14732.493,E2 14732.493} C_VEL
LIN {X 0,Y 550.778,Z 483.24,A -85,B 0,C 180,E1 14730.11,E2 14730.11} C_VEL
LIN {X 0,Y 540.034,Z 694.836,A -85,B 0,C 180,E1 14726.88,E2 14726.88} C_VEL
LIN {X 0,Y 533.486,Z 825.698,A -85,B 0,C 180,E1 14724.88,E2 14724.88} C_VEL
LIN {X 0,Y 531.023,Z 852.911,A -85,B 0,C 180,E1 14724.363,E2 14724.363} C_VEL
LIN {X 0,Y 527.541,Z 879.572,A -85,B 0,C 180,E1 14723.667,E2 14723.667} C_VEL
LIN {X 0,Y 524.177,Z 901.088,A -85,B 0,C 180,E1 14722.968,E2 14722.968} C_VEL
LIN {X 0,Y 520.546,Z 921.382,A -85,B 0,C 180,E1 14722.18,E2 14722.18} C_VEL
LIN {X 0,Y 516.289,Z 942.551,A -85,B 0,C 180,E1 14721.216,E2 14721.216} C_VEL
LIN {X 0,Y 510.697,Z 967.605,A -85,B 0,C 180,E1 14719.867,E2 14719.867} C_VEL
LIN {X 0,Y 504.878,Z 990.707,A -85,B 0,C 180,E1 14718.384,E2 14718.384} C_VEL
LIN {X 0,Y 499.997,Z 1008.898,A -85,B 0,C 180,E1 14717.048,E2 14717.048} C_VEL
LIN {X 0,Y 495.142,Z 1026.019,A -85,B 0,C 180,E1 14715.632,E2 14715.632} C_VEL
LIN {X 0,Y 489.994,Z 1043.432,A -85,B 0,C 180,E1 14714.013,E2 14714.013} C_VEL
LIN {X 0,Y 483.852,Z 1063.716,A -85,B 0,C 180,E1 14711.873,E2 14711.873} C_VEL
LIN {X 0,Y 477.763,Z 1082.971,A -85,B 0,C 180,E1 14709.511,E2 14709.511} C_VEL
LIN {X 0,Y 472.805,Z 1098.626,A -85,B 0,C 180,E1 14707.329,E2 14707.329} C_VEL
LIN {X 0,Y 468.251,Z 1113.104,A -85,B 0,C 180,E1 14705.059,E2 14705.059} C_VEL
LIN {X 0,Y 463.563,Z 1128.445,A -85,B 0,C 180,E1 14702.339,E2 14702.339} C_VEL
LIN {X 0,Y 459.11,Z 1143.614,A -85,B 0,C 180,E1 14699.199,E2 14699.199} C_VEL
LIN {X 0,Y 456.077,Z 1154.735,A -85,B 0,C 180,E1 14696.557,E2 14696.557} C_VEL
LIN {X 0,Y 453.656,Z 1164.498,A -85,B 0,C 180,E1 14693.926,E2 14693.926} C_VEL
LIN {X 0,Y 451.674,Z 1173.513,A -85,B 0,C 180,E1 14691.152,E2 14691.152} C_VEL
LIN {X 0,Y 449.926,Z 1183.004,A -85,B 0,C 180,E1 14687.726,E2 14687.726} C_VEL
LIN {X 0,Y 448.906,Z 1190.042,A -85,B 0,C 180,E1 14684.578,E2 14684.578} C_VEL
LIN {X 0,Y 448.344,Z 1195.214,A -85,B 0,C 180,E1 14681.747,E2 14681.747} C_VEL
LIN {X 0,Y 448.078,Z 1199.022,A -85,B 0,C 180,E1 14679.117,E2 14679.117} C_VEL
LIN {X 0,Y 447.961,Z 1201.825,A -85,B 0,C 180,E1 14676.537,E2 14676.537} C_VEL
LIN {X 0,Y 447.915,Z 1203.7,A -85,B 0,C 180,E1 14673.969,E2 14673.969} C_VEL
LIN {X 0,Y 447.912,Z 1204.658,A -85,B 0,C 180,E1 14671.408,E2 14671.408} C_VEL
LIN {X 0,Y 447.912,Z 1204.703,A -85,B 0,C 180,E1 14668.849,E2 14668.849} C_VEL
LIN {X 0,Y 447.914,Z 1203.813,A -85,B 0,C 180,E1 14666.247,E2 14666.247} C_VEL
LIN {X 0,Y 447.953,Z 1202.052,A -85,B 0,C 180,E1 14663.721,E2 14663.721} C_VEL
LIN {X 0,Y 448.063,Z 1199.341,A -85,B 0,C 180,E1 14661.143,E2 14661.143} C_VEL
LIN {X 0,Y 448.298,Z 1195.686,A -85,B 0,C 180,E1 14658.551,E2 14658.551} C_VEL
LIN {X 0,Y 448.813,Z 1190.806,A -85,B 0,C 180,E1 14655.815,E2 14655.815} C_VEL
LIN {X 0,Y 449.614,Z 1184.827,A -85,B 0,C 180,E1 14653.063,E2 14653.063} C_VEL
LIN {X 0,Y 451.14,Z 1176.285,A -85,B 0,C 180,E1 14649.773,E2 14649.773} C_VEL
LIN {X 0,Y 453.444,Z 1165.402,A -85,B 0,C 180,E1 14646.34,E2 14646.34} C_VEL
LIN {X 0,Y 455.82,Z 1155.708,A -85,B 0,C 180,E1 14643.699,E2 14643.699} C_VEL
LIN {X 0,Y 458.766,Z 1144.761,A -85,B 0,C 180,E1 14641.064,E2 14641.064} C_VEL
LIN {X 0,Y 462.789,Z 1131.217,A -85,B 0,C 180,E1 14638.186,E2 14638.186} C_VEL
LIN {X 0,Y 468.058,Z 1114.244,A -85,B 0,C 180,E1 14635.075,E2 14635.075} C_VEL
LIN {X 0,Y 472.702,Z 1099.916,A -85,B 0,C 180,E1 14632.775,E2 14632.775} C_VEL
LIN {X 0,Y 477.617,Z 1084.957,A -85,B 0,C 180,E1 14630.631,E2 14630.631} C_VEL
LIN {X 0,Y 483.257,Z 1067.916,A -85,B 0,C 180,E1 14628.462,E2 14628.462} C_VEL
LIN {X 0,Y 490.57,Z 1045.317,A -85,B 0,C 180,E1 14625.972,E2 14625.972} C_VEL
LIN {X 0,Y 496.424,Z 1026.603,A -85,B 0,C 180,E1 14624.19,E2 14624.19} C_VEL
LIN {X 0,Y 501.639,Z 1009.329,A -85,B 0,C 180,E1 14622.736,E2 14622.736} C_VEL
LIN {X 0,Y 506.924,Z 990.893,A -85,B 0,C 180,E1 14621.359,E2 14621.359} C_VEL
LIN {X 0,Y 512.432,Z 970.414,A -85,B 0,C 180,E1 14620.017,E2 14620.017} C_VEL
LIN {X 0,Y 518.957,Z 943.629,A -85,B 0,C 180,E1 14618.535,E2 14618.535} C_VEL
LIN {X 0,Y 523.712,Z 921.653,A -85,B 0,C 180,E1 14617.521,E2 14617.521} C_VEL
LIN {X 0,Y 527.646,Z 901.216,A -85,B 0,C 180,E1 14616.72,E2 14616.72} C_VEL
LIN {X 0,Y 531.277,Z 879.66,A -85,B 0,C 180,E1 14616.016,E2 14616.016} C_VEL
LIN {X 0,Y 534.854,Z 854.29,A -85,B 0,C 180,E1 14615.348,E2 14615.348} C_VEL
LIN {X 0,Y 537.66,Z 826.353,A -85,B 0,C 180,E1 14614.806,E2 14614.806} C_VEL
LIN {X 0,Y 542.825,Z 735.776,A -85,B 0,C 180,E1 14613.395,E2 14613.395} C_VEL
LIN {X 0,Y 555.299,Z 518.548,A -85,B 0,C 180,E1 14610.036,E2 14610.036} C_VEL
LIN {X 0,Y 557.297,Z 484.972,A -85,B 0,C 180,E1 14609.511,E2 14609.511} C_VEL
LIN {X 0,Y 547.294,Z 469.147,A -85,B 0,C 180,E1 14606.913,E2 14606.913} C_VEL
LIN {X 0,Y 538.39,Z 456.101,A -85,B 0,C 180,E1 14604.291,E2 14604.291} C_VEL
LIN {X 0,Y 532.403,Z 447.708,A -85,B 0,C 180,E1 14602.295,E2 14602.295} C_VEL
LIN {X 0,Y 528.415,Z 442.62,A -85,B 0,C 180,E1 14600.839,E2 14600.839} C_VEL
LIN {X 0,Y 524.228,Z 437.328,A -85,B 0,C 180,E1 14599.151,E2 14599.151} C_VEL
LIN {X 0,Y 520.685,Z 432.785,A -85,B 0,C 180,E1 14597.547,E2 14597.547} C_VEL
LIN {X 0,Y 516.201,Z 427.49,A -85,B 0,C 180,E1 14595.217,E2 14595.217} C_VEL
LIN {X 0,Y 515.396,Z 426.189,A -85,B 0,C 180,E1 14594.723,E2 14594.723} C_VEL
LIN {X 0,Y 512.214,Z 423.226,A -85,B 0,C 180,E1 14592.686,E2 14592.686} C_VEL
LIN {X 0,Y 510.44,Z 420.029,A -85,B 0,C 180,E1 14591.182,E2 14591.182} C_VEL
LIN {X 0,Y 506.823,Z 416.928,A -85,B 0,C 180,E1 14587.14,E2 14587.14} C_VEL
LIN {X 0,Y 505.838,Z 413.72,A -85,B 0,C 180,E1 14583.627,E2 14583.627} C_VEL
LIN {X 0,Y 505.87,Z 413.89,A -85,B 0,C 180,E1 14581.812,E2 14581.812} C_VEL
LIN {X 0,Y 508.933,Z 419.181,A -85,B 0,C 180,E1 14575.944,E2 14575.944} C_VEL
LIN {X 0,Y 510.706,Z 420.379,A -85,B 0,C 180,E1 14574.382,E2 14574.382} C_VEL
LIN {X 0,Y 512.917,Z 424.062,A -85,B 0,C 180,E1 14572.608,E2 14572.608} C_VEL
LIN {X 0,Y 515.76,Z 426.677,A -85,B 0,C 180,E1 14570.853,E2 14570.853} C_VEL
LIN {X 0,Y 518.774,Z 430.872,A -85,B 0,C 180,E1 14569.168,E2 14569.168} C_VEL
LIN {X 0,Y 520.68,Z 432.693,A -85,B 0,C 180,E1 14568.255,E2 14568.255} C_VEL
LIN {X 0,Y 524.463,Z 437.483,A -85,B 0,C 180,E1 14566.55,E2 14566.55} C_VEL
LIN {X 0,Y 530.325,Z 444.97,A -85,B 0,C 180,E1 14564.246,E2 14564.246} C_VEL
LIN {X 0,Y 534.901,Z 450.846,A -85,B 0,C 180,E1 14562.653,E2 14562.653} C_VEL
LIN {X 0,Y 541.493,Z 459.475,A -85,B 0,C 180,E1 14560.587,E2 14560.587} C_VEL
LIN {X 0,Y 550.857,Z 472.441,A -85,B 0,C 180,E1 14557.986,E2 14557.986} C_VEL
LIN {X 0,Y 557.094,Z 482.042,A -85,B 0,C 180,E1 14556.406,E2 14556.406} C_VEL
LIN {X 0,Y 557.299,Z 482.839,A -85,B 0,C 180,E1 14556.343,E2 14556.343} C_VEL
LIN {X 0,Y 544.755,Z 698.073,A -85,B 0,C 180,E1 14553.013,E2 14553.013} C_VEL
LIN {X 0,Y 537.872,Z 819.222,A -85,B 0,C 180,E1 14551.131,E2 14551.131} C_VEL
LIN {X 0,Y 535.219,Z 846.462,A -85,B 0,C 180,E1 14550.605,E2 14550.605} C_VEL
LIN {X 0,Y 531.531,Z 872.902,A -85,B 0,C 180,E1 14549.904,E2 14549.904} C_VEL
LIN {X 0,Y 528.071,Z 893.689,A -85,B 0,C 180,E1 14549.22,E2 14549.22} C_VEL
LIN {X 0,Y 524.256,Z 913.712,A -85,B 0,C 180,E1 14548.435,E2 14548.435} C_VEL
LIN {X 0,Y 519.868,Z 934.135,A -85,B 0,C 180,E1 14547.498,E2 14547.498} C_VEL
LIN {X 0,Y 514.517,Z 956.802,A -85,B 0,C 180,E1 14546.277,E2 14546.277} C_VEL
LIN {X 0,Y 507.893,Z 981.673,A -85,B 0,C 180,E1 14544.687,E2 14544.687} C_VEL
LIN {X 0,Y 502.542,Z 1000.312,A -85,B 0,C 180,E1 14543.304,E2 14543.304} C_VEL
LIN {X 0,Y 497.238,Z 1017.815,A -85,B 0,C 180,E1 14541.835,E2 14541.835} C_VEL
LIN {X 0,Y 491.655,Z 1035.486,A -85,B 0,C 180,E1 14540.161,E2 14540.161} C_VEL
LIN {X 0,Y 485.604,Z 1054.172,A -85,B 0,C 180,E1 14538.153,E2 14538.153} C_VEL
LIN {X 0,Y 478.711,Z 1074.78,A -85,B 0,C 180,E1 14535.587,E2 14535.587} C_VEL
LIN {X 0,Y 473.434,Z 1090.489,A -85,B 0,C 180,E1 14533.344,E2 14533.344} C_VEL
LIN {X 0,Y 468.743,Z 1104.645,A -85,B 0,C 180,E1 14531.07,E2 14531.07} C_VEL
LIN {X 0,Y 463.764,Z 1120.31,A -85,B 0,C 180,E1 14528.226,E2 14528.226} C_VEL
LIN {X 0,Y 459.229,Z 1135.12,A -85,B 0,C 180,E1 14525.085,E2 14525.085} C_VEL
LIN {X 0,Y 456.16,Z 1146.04,A -85,B 0,C 180,E1 14522.444,E2 14522.444} C_VEL
LIN {X 0,Y 453.757,Z 1155.453,A -85,B 0,C 180,E1 14519.867,E2 14519.867} C_VEL
LIN {X 0,Y 451.898,Z 1163.599,A -85,B 0,C 180,E1 14517.332,E2 14517.332} C_VEL
LIN {X 0,Y 450.362,Z 1166.478,A -85,B 0,C 180,E1 14516.434,E2 14516.434} C_VEL
LIN {X 0,Y 442.777,Z 1173.71,A -85,B 0,C 180,E1 14513.978,E2 14513.978} C_VEL
LIN {X 0,Y 441.817,Z 1175.453,A -85,B 0,C 180,E1 14513.23,E2 14513.23} C_VEL
LIN {X 0,Y 440.911,Z 1181.309,A -85,B 0,C 180,E1 14510.44,E2 14510.44} C_VEL
LIN {X 0,Y 440.376,Z 1186.015,A -85,B 0,C 180,E1 14507.712,E2 14507.712} C_VEL
LIN {X 0,Y 440.087,Z 1189.703,A -85,B 0,C 180,E1 14505.011,E2 14505.011} C_VEL
LIN {X 0,Y 439.956,Z 1192.411,A -85,B 0,C 180,E1 14502.335,E2 14502.335} C_VEL
LIN {X 0,Y 439.917,Z 1194.171,A -85,B 0,C 180,E1 14499.682,E2 14499.682} C_VEL
LIN {X 0,Y 439.905,Z 1195.006,A -85,B 0,C 180,E1 14497.05,E2 14497.05} C_VEL
LIN {X 0,Y 439.91,Z 1194.91,A -85,B 0,C 180,E1 14494.301,E2 14494.301} C_VEL
LIN {X 0,Y 439.922,Z 1193.761,A -85,B 0,C 180,E1 14491.432,E2 14491.432} C_VEL
LIN {X 0,Y 440.016,Z 1191.076,A -85,B 0,C 180,E1 14488.046,E2 14488.046} C_VEL
LIN {X 0,Y 440.3,Z 1186.717,A -85,B 0,C 180,E1 14484.657,E2 14484.657} C_VEL
LIN {X 0,Y 440.843,Z 1181.892,A -85,B 0,C 180,E1 14481.784,E2 14481.784} C_VEL
LIN {X 0,Y 441.67,Z 1176.242,A -85,B 0,C 180,E1 14479.037,E2 14479.037} C_VEL
LIN {X 0,Y 442.914,Z 1169.533,A -85,B 0,C 180,E1 14476.288,E2 14476.288} C_VEL
LIN {X 0,Y 444.839,Z 1160.841,A -85,B 0,C 180,E1 14473.246,E2 14473.246} C_VEL
LIN {X 0,Y 448.046,Z 1148.422,A -85,B 0,C 180,E1 14469.604,E2 14469.604} C_VEL
LIN {X 0,Y 451.114,Z 1137.64,A -85,B 0,C 180,E1 14466.901,E2 14466.901} C_VEL
LIN {X 0,Y 454.716,Z 1125.986,A -85,B 0,C 180,E1 14464.33,E2 14464.33} C_VEL
LIN {X 0,Y 458.914,Z 1112.935,A -85,B 0,C 180,E1 14461.784,E2 14461.784} C_VEL
LIN {X 0,Y 464.789,Z 1095.166,A -85,B 0,C 180,E1 14458.771,E2 14458.771} C_VEL
LIN {X 0,Y 470.121,Z 1079.142,A -85,B 0,C 180,E1 14456.428,E2 14456.428} C_VEL
LIN {X 0,Y 475.21,Z 1063.741,A -85,B 0,C 180,E1 14454.428,E2 14454.428} C_VEL
LIN {X 0,Y 480.608,Z 1047.172,A -85,B 0,C 180,E1 14452.516,E2 14452.516} C_VEL
LIN {X 0,Y 487.407,Z 1025.814,A -85,B 0,C 180,E1 14450.357,E2 14450.357} C_VEL
LIN {X 0,Y 493.691,Z 1004.564,A -85,B 0,C 180,E1 14448.526,E2 14448.526} C_VEL
LIN {X 0,Y 498.878,Z 986.012,A -85,B 0,C 180,E1 14447.121,E2 14447.121} C_VEL
LIN {X 0,Y 503.872,Z 966.944,A -85,B 0,C 180,E1 14445.851,E2 14445.851} C_VEL
LIN {X 0,Y 509.103,Z 945.401,A -85,B 0,C 180,E1 14444.606,E2 14444.606} C_VEL
LIN {X 0,Y 514.759,Z 919.141,A -85,B 0,C 180,E1 14443.328,E2 14443.328} C_VEL
LIN {X 0,Y 518.898,Z 896.993,A -85,B 0,C 180,E1 14442.437,E2 14442.437} C_VEL
LIN {X 0,Y 522.347,Z 875.653,A -85,B 0,C 180,E1 14441.719,E2 14441.719} C_VEL
LIN {X 0,Y 525.265,Z 854.328,A -85,B 0,C 180,E1 14441.13,E2 14441.13} C_VEL
LIN {X 0,Y 527.863,Z 830.744,A -85,B 0,C 180,E1 14440.615,E2 14440.615} C_VEL
LIN {X 0,Y 530.243,Z 794.735,A -85,B 0,C 180,E1 14440.021,E2 14440.021} C_VEL
LIN {X 0,Y 541.662,Z 571.918,A -85,B 0,C 180,E1 14436.622,E2 14436.622} C_VEL
LIN {X 0,Y 546.285,Z 484.636,A -85,B 0,C 180,E1 14435.273,E2 14435.273} C_VEL
LIN {X 0,Y 538.307,Z 472.539,A -85,B 0,C 180,E1 14433.546,E2 14433.546} C_VEL
LIN {X 0,Y 528.724,Z 459.131,A -85,B 0,C 180,E1 14431.305,E2 14431.305} C_VEL
LIN {X 0,Y 519.158,Z 446.114,A -85,B 0,C 180,E1 14428.815,E2 14428.815} C_VEL
LIN {X 0,Y 510.124,Z 434.6,A -85,B 0,C 180,E1 14426.169,E2 14426.169} C_VEL
LIN {X 0,Y 505.675,Z 429.026,A -85,B 0,C 180,E1 14424.722,E2 14424.722} C_VEL
LIN {X 0,Y 501.502,Z 423.853,A -85,B 0,C 180,E1 14423.252,E2 14423.252} C_VEL
LIN {X 0,Y 496.915,Z 418.301,A -85,B 0,C 180,E1 14421.483,E2 14421.483} C_VEL
LIN {X 0,Y 493.227,Z 413.987,A -85,B 0,C 180,E1 14419.912,E2 14419.912} C_VEL
LIN {X 0,Y 492.262,Z 412.583,A -85,B 0,C 180,E1 14419.458,E2 14419.458} C_VEL
LIN {X 0,Y 488.82,Z 409.141,A -85,B 0,C 180,E1 14417.807,E2 14417.807} C_VEL
LIN {X 0,Y 487.282,Z 406.656,A -85,B 0,C 180,E1 14416.941,E2 14416.941} C_VEL
LIN {X 0,Y 483.711,Z 403.5,A -85,B 0,C 180,E1 14414.852,E2 14414.852} C_VEL
LIN {X 0,Y 481.823,Z 400.201,A -85,B 0,C 180,E1 14413.44,E2 14413.44} C_VEL
LIN {X 0,Y 478.203,Z 397.496,A -85,B 0,C 180,E1 14410.359,E2 14410.359} C_VEL
LIN {X 0,Y 476.639,Z 394.056,A -85,B 0,C 180,E1 14408.141,E2 14408.141} C_VEL
LIN {X 0,Y 474.925,Z 393.294,A -85,B 0,C 180,E1 14403.742,E2 14403.742} C_VEL
LIN {X 0,Y 476.583,Z 393.851,A -85,B 0,C 180,E1 14398.076,E2 14398.076} C_VEL
LIN {X 0,Y 478.362,Z 397.765,A -85,B 0,C 180,E1 14395.564,E2 14395.564} C_VEL
LIN {X 0,Y 482.124,Z 400.639,A -85,B 0,C 180,E1 14392.432,E2 14392.432} C_VEL
LIN {X 0,Y 484.685,Z 404.721,A -85,B 0,C 180,E1 14390.62,E2 14390.62} C_VEL
LIN {X 0,Y 487.558,Z 407.076,A -85,B 0,C 180,E1 14389.005,E2 14389.005} C_VEL
LIN {X 0,Y 490.477,Z 411.12,A -85,B 0,C 180,E1 14387.461,E2 14387.461} C_VEL
LIN {X 0,Y 492.818,Z 413.298,A -85,B 0,C 180,E1 14386.387,E2 14386.387} C_VEL
LIN {X 0,Y 496.122,Z 417.694,A -85,B 0,C 180,E1 14384.931,E2 14384.931} C_VEL
LIN {X 0,Y 498.002,Z 419.644,A -85,B 0,C 180,E1 14384.183,E2 14384.183} C_VEL
LIN {X 0,Y 501.839,Z 424.244,A -85,B 0,C 180,E1 14382.73,E2 14382.73} C_VEL
LIN {X 0,Y 507.691,Z 431.665,A -85,B 0,C 180,E1 14380.708,E2 14380.708} C_VEL
LIN {X 0,Y 512.672,Z 437.916,A -85,B 0,C 180,E1 14379.149,E2 14379.149} C_VEL
LIN {X 0,Y 519.161,Z 446.253,A -85,B 0,C 180,E1 14377.284,E2 14377.284} C_VEL
LIN {X 0,Y 528.262,Z 459.52,A -85,B 0,C 180,E1 14374.883,E2 14374.883} C_VEL
LIN {X 0,Y 536.879,Z 472.664,A -85,B 0,C 180,E1 14372.822,E2 14372.822} C_VEL
LIN {X 0,Y 546.303,Z 487.522,A -85,B 0,C 180,E1 14370.757,E2 14370.757} C_VEL
LIN {X 0,Y 535.175,Z 699.825,A -85,B 0,C 180,E1 14367.504,E2 14367.504} C_VEL
LIN {X 0,Y 528.659,Z 825.695,A -85,B 0,C 180,E1 14365.572,E2 14365.572} C_VEL
LIN {X 0,Y 526.114,Z 853.076,A -85,B 0,C 180,E1 14365.05,E2 14365.05} C_VEL
LIN {X 0,Y 522.56,Z 879.574,A -85,B 0,C 180,E1 14364.358,E2 14364.358} C_VEL
LIN {X 0,Y 519.135,Z 900.898,A -85,B 0,C 180,E1 14363.666,E2 14363.666} C_VEL
LIN {X 0,Y 515.405,Z 921.205,A -85,B 0,C 180,E1 14362.877,E2 14362.877} C_VEL
LIN {X 0,Y 511.169,Z 941.694,A -85,B 0,C 180,E1 14361.945,E2 14361.945} C_VEL
LIN {X 0,Y 505.635,Z 966.072,A -85,B 0,C 180,E1 14360.642,E2 14360.642} C_VEL
LIN {X 0,Y 499.615,Z 989.346,A -85,B 0,C 180,E1 14359.156,E2 14359.156} C_VEL
LIN {X 0,Y 494.55,Z 1007.662,A -85,B 0,C 180,E1 14357.816,E2 14357.816} C_VEL
LIN {X 0,Y 489.201,Z 1025.945,A -85,B 0,C 180,E1 14356.303,E2 14356.303} C_VEL
LIN {X 0,Y 483.789,Z 1043.655,A -85,B 0,C 180,E1 14354.644,E2 14354.644} C_VEL
LIN {X 0,Y 477.263,Z 1064.483,A -85,B 0,C 180,E1 14352.423,E2 14352.423} C_VEL
LIN {X 0,Y 470.968,Z 1083.619,A -85,B 0,C 180,E1 14350.037,E2 14350.037} C_VEL
LIN {X 0,Y 465.912,Z 1098.997,A -85,B 0,C 180,E1 14347.863,E2 14347.863} C_VEL
LIN {X 0,Y 461.307,Z 1113.076,A -85,B 0,C 180,E1 14345.627,E2 14345.627} C_VEL
LIN {X 0,Y 456.242,Z 1128.965,A -85,B 0,C 180,E1 14342.773,E2 14342.773} C_VEL
LIN {X 0,Y 451.793,Z 1143.475,A -85,B 0,C 180,E1 14339.719,E2 14339.719} C_VEL
LIN {X 0,Y 448.598,Z 1154.591,A -85,B 0,C 180,E1 14337.046,E2 14337.046} C_VEL
LIN {X 0,Y 446.032,Z 1164.405,A -85,B 0,C 180,E1 14334.361,E2 14334.361} C_VEL
LIN {X 0,Y 443.925,Z 1173.455,A -85,B 0,C 180,E1 14331.528,E2 14331.528} C_VEL
LIN {X 0,Y 442.009,Z 1183.22,A -85,B 0,C 180,E1 14327.918,E2 14327.918} C_VEL
LIN {X 0,Y 440.944,Z 1190.21,A -85,B 0,C 180,E1 14324.713,E2 14324.713} C_VEL
LIN {X 0,Y 440.366,Z 1195.276,A -85,B 0,C 180,E1 14321.867,E2 14321.867} C_VEL
LIN {X 0,Y 440.09,Z 1198.934,A -85,B 0,C 180,E1 14319.283,E2 14319.283} C_VEL
LIN {X 0,Y 439.962,Z 1201.737,A -85,B 0,C 180,E1 14316.656,E2 14316.656} C_VEL
LIN {X 0,Y 439.915,Z 1203.612,A -85,B 0,C 180,E1 14314.041,E2 14314.041} C_VEL
LIN {X 0,Y 439.912,Z 1204.571,A -85,B 0,C 180,E1 14311.433,E2 14311.433} C_VEL
LIN {X 0,Y 439.912,Z 1204.616,A -85,B 0,C 180,E1 14308.828,E2 14308.828} C_VEL
LIN {X 0,Y 439.914,Z 1203.744,A -85,B 0,C 180,E1 14306.214,E2 14306.214} C_VEL
LIN {X 0,Y 439.957,Z 1201.963,A -85,B 0,C 180,E1 14303.607,E2 14303.607} C_VEL
LIN {X 0,Y 440.074,Z 1199.251,A -85,B 0,C 180,E1 14300.981,E2 14300.981} C_VEL
LIN {X 0,Y 440.33,Z 1195.595,A -85,B 0,C 180,E1 14298.341,E2 14298.341} C_VEL
LIN {X 0,Y 440.875,Z 1190.732,A -85,B 0,C 180,E1 14295.564,E2 14295.564} C_VEL
LIN {X 0,Y 441.744,Z 1184.733,A -85,B 0,C 180,E1 14292.752,E2 14292.752} C_VEL
LIN {X 0,Y 443.373,Z 1176.118,A -85,B 0,C 180,E1 14289.376,E2 14289.376} C_VEL
LIN {X 0,Y 445.809,Z 1165.282,A -85,B 0,C 180,E1 14285.902,E2 14285.902} C_VEL
LIN {X 0,Y 448.429,Z 1155.211,A -85,B 0,C 180,E1 14283.114,E2 14283.114} C_VEL
LIN {X 0,Y 451.517,Z 1144.489,A -85,B 0,C 180,E1 14280.495,E2 14280.495} C_VEL
LIN {X 0,Y 455.862,Z 1130.581,A -85,B 0,C 180,E1 14277.495,E2 14277.495} C_VEL
LIN {X 0,Y 461.212,Z 1114.294,A -85,B 0,C 180,E1 14274.479,E2 14274.479} C_VEL
LIN {X 0,Y 466.113,Z 1099.861,A -85,B 0,C 180,E1 14272.132,E2 14272.132} C_VEL
LIN {X 0,Y 471.195,Z 1085.073,A -85,B 0,C 180,E1 14269.987,E2 14269.987} C_VEL
LIN {X 0,Y 476.6,Z 1069.38,A -85,B 0,C 180,E1 14267.961,E2 14267.961} C_VEL
LIN {X 0,Y 483.52,Z 1049.15,A -85,B 0,C 180,E1 14265.658,E2 14265.658} C_VEL
LIN {X 0,Y 490.308,Z 1028.186,A -85,B 0,C 180,E1 14263.62,E2 14263.62} C_VEL
LIN {X 0,Y 495.897,Z 1010.365,A -85,B 0,C 180,E1 14262.099,E2 14262.099} C_VEL
LIN {X 0,Y 501.095,Z 992.921,A -85,B 0,C 180,E1 14260.779,E2 14260.779} C_VEL
LIN {X 0,Y 506.273,Z 974.381,A -85,B 0,C 180,E1 14259.537,E2 14259.537} C_VEL
LIN {X 0,Y 511.698,Z 953.546,A -85,B 0,C 180,E1 14258.322,E2 14258.322} C_VEL
LIN {X 0,Y 517.844,Z 927.32,A -85,B 0,C 180,E1 14257.032,E2 14257.032} C_VEL
LIN {X 0,Y 522.623,Z 903.59,A -85,B 0,C 180,E1 14256.078,E2 14256.078} C_VEL
LIN {X 0,Y 526.382,Z 882.198,A -85,B 0,C 180,E1 14255.365,E2 14255.365} C_VEL
LIN {X 0,Y 529.518,Z 861.094,A -85,B 0,C 180,E1 14254.788,E2 14254.788} C_VEL
LIN {X 0,Y 532.374,Z 837.4,A -85,B 0,C 180,E1 14254.277,E2 14254.277} C_VEL
LIN {X 0,Y 534.991,Z 801.406,A -85,B 0,C 180,E1 14253.677,E2 14253.677} C_VEL
LIN {X 0,Y 547.861,Z 579.881,A -85,B 0,C 180,E1 14250.251,E2 14250.251} C_VEL
LIN {X 0,Y 553.372,Z 489.685,A -85,B 0,C 180,E1 14248.845,E2 14248.845} C_VEL
LIN {X 0,Y 544.184,Z 474.974,A -85,B 0,C 180,E1 14246.372,E2 14246.372} C_VEL
LIN {X 0,Y 535.735,Z 462.528,A -85,B 0,C 180,E1 14243.804,E2 14243.804} C_VEL
LIN {X 0,Y 530.552,Z 455.094,A -85,B 0,C 180,E1 14242.027,E2 14242.027} C_VEL
LIN {X 0,Y 526.764,Z 450.178,A -85,B 0,C 180,E1 14240.617,E2 14240.617} C_VEL
LIN {X 0,Y 522.639,Z 444.906,A -85,B 0,C 180,E1 14238.922,E2 14238.922} C_VEL
LIN {X 0,Y 519.052,Z 440.163,A -85,B 0,C 180,E1 14237.257,E2 14237.257} C_VEL
LIN {X 0,Y 514.942,Z 435.353,A -85,B 0,C 180,E1 14235.082,E2 14235.082} C_VEL
LIN {X 0,Y 514.056,Z 433.96,A -85,B 0,C 180,E1 14234.532,E2 14234.532} C_VEL
LIN {X 0,Y 510.875,Z 430.818,A -85,B 0,C 180,E1 14232.433,E2 14232.433} C_VEL
LIN {X 0,Y 509.34,Z 427.929,A -85,B 0,C 180,E1 14231.092,E2 14231.092} C_VEL
LIN {X 0,Y 505.785,Z 424.812,A -85,B 0,C 180,E1 14227.04,E2 14227.04} C_VEL
LIN {X 0,Y 504.85,Z 421.665,A -85,B 0,C 180,E1 14223.52,E2 14223.52} C_VEL
LIN {X 0,Y 504.887,Z 421.881,A -85,B 0,C 180,E1 14221.816,E2 14221.816} C_VEL
LIN {X 0,Y 507.955,Z 427.142,A -85,B 0,C 180,E1 14215.936,E2 14215.936} C_VEL
LIN {X 0,Y 509.58,Z 428.346,A -85,B 0,C 180,E1 14214.483,E2 14214.483} C_VEL
LIN {X 0,Y 511.933,Z 432.123,A -85,B 0,C 180,E1 14212.593,E2 14212.593} C_VEL
LIN {X 0,Y 514.487,Z 434.535,A -85,B 0,C 180,E1 14210.999,E2 14210.999} C_VEL
LIN {X 0,Y 517.577,Z 438.766,A -85,B 0,C 180,E1 14209.256,E2 14209.256} C_VEL
LIN {X 0,Y 519.344,Z 440.579,A -85,B 0,C 180,E1 14208.393,E2 14208.393} C_VEL
LIN {X 0,Y 523.229,Z 445.392,A -85,B 0,C 180,E1 14206.63,E2 14206.63} C_VEL
LIN {X 0,Y 528.758,Z 452.706,A -85,B 0,C 180,E1 14204.423,E2 14204.423} C_VEL
LIN {X 0,Y 533.133,Z 458.395,A -85,B 0,C 180,E1 14202.875,E2 14202.875} C_VEL
LIN {X 0,Y 539.56,Z 466.965,A -85,B 0,C 180,E1 14200.824,E2 14200.824} C_VEL
LIN {X 0,Y 548.822,Z 479.923,A -85,B 0,C 180,E1 14198.21,E2 14198.21} C_VEL
LIN {X 0,Y 553.396,Z 487.089,A -85,B 0,C 180,E1 14197.02,E2 14197.02} C_VEL
LIN {X 0,Y 540.746,Z 697.39,A -85,B 0,C 180,E1 14193.756,E2 14193.756} C_VEL
LIN {X 0,Y 533.585,Z 819.342,A -85,B 0,C 180,E1 14191.857,E2 14191.857} C_VEL
LIN {X 0,Y 530.844,Z 846.709,A -85,B 0,C 180,E1 14191.327,E2 14191.327} C_VEL
LIN {X 0,Y 527.079,Z 872.974,A -85,B 0,C 180,E1 14190.632,E2 14190.632} C_VEL
LIN {X 0,Y 523.544,Z 893.621,A -85,B 0,C 180,E1 14189.955,E2 14189.955} C_VEL
LIN {X 0,Y 519.633,Z 913.612,A -85,B 0,C 180,E1 14189.172,E2 14189.172} C_VEL
LIN {X 0,Y 515.103,Z 934.112,A -85,B 0,C 180,E1 14188.233,E2 14188.233} C_VEL
LIN {X 0,Y 509.842,Z 955.725,A -85,B 0,C 180,E1 14187.073,E2 14187.073} C_VEL
LIN {X 0,Y 503.069,Z 980.592,A -85,B 0,C 180,E1 14185.496,E2 14185.496} C_VEL
LIN {X 0,Y 497.244,Z 1000.2,A -85,B 0,C 180,E1 14184.043,E2 14184.043} C_VEL
LIN {X 0,Y 491.675,Z 1017.931,A -85,B 0,C 180,E1 14182.551,E2 14182.551} C_VEL
LIN {X 0,Y 485.904,Z 1035.541,A -85,B 0,C 180,E1 14180.875,E2 14180.875} C_VEL
LIN {X 0,Y 479.359,Z 1054.998,A -85,B 0,C 180,E1 14178.765,E2 14178.765} C_VEL
LIN {X 0,Y 472.298,Z 1075.219,A -85,B 0,C 180,E1 14176.212,E2 14176.212} C_VEL
LIN {X 0,Y 466.87,Z 1090.679,A -85,B 0,C 180,E1 14173.978,E2 14173.978} C_VEL
LIN {X 0,Y 461.91,Z 1104.992,A -85,B 0,C 180,E1 14171.647,E2 14171.647} C_VEL
LIN {X 0,Y 456.678,Z 1120.608,A -85,B 0,C 180,E1 14168.768,E2 14168.768} C_VEL
LIN {X 0,Y 451.921,Z 1135.353,A -85,B 0,C 180,E1 14165.583,E2 14165.583} C_VEL
LIN {X 0,Y 448.716,Z 1146.098,A -85,B 0,C 180,E1 14162.936,E2 14162.936} C_VEL
LIN {X 0,Y 446.136,Z 1155.608,A -85,B 0,C 180,E1 14160.282,E2 14160.282} C_VEL
LIN {X 0,Y 443.94,Z 1164.793,A -85,B 0,C 180,E1 14157.352,E2 14157.352} C_VEL
LIN {X 0,Y 441.97,Z 1174.611,A -85,B 0,C 180,E1 14153.604,E2 14153.604} C_VEL
LIN {X 0,Y 441.817,Z 1175.453,A -85,B 0,C 180,E1 14153.23,E2 14153.23} C_VEL
LIN {X 0,Y 440.458,Z 1177.694,A -85,B 0,C 180,E1 14152.279,E2 14152.279} C_VEL
LIN {X 0,Y 433.374,Z 1183.344,A -85,B 0,C 180,E1 14149.674,E2 14149.674} C_VEL
LIN {X 0,Y 432.575,Z 1184.656,A -85,B 0,C 180,E1 14148.889,E2 14148.889} C_VEL
LIN {X 0,Y 432.156,Z 1189.172,A -85,B 0,C 180,E1 14145.705,E2 14145.705} C_VEL
LIN {X 0,Y 431.977,Z 1192.176,A -85,B 0,C 180,E1 14142.838,E2 14142.838} C_VEL
LIN {X 0,Y 431.921,Z 1194.067,A -85,B 0,C 180,E1 14140.133,E2 14140.133} C_VEL
LIN {X 0,Y 431.915,Z 1195.03,A -85,B 0,C 180,E1 14137.448,E2 14137.448} C_VEL
LIN {X 0,Y 431.904,Z 1195.083,A -85,B 0,C 180,E1 14134.78,E2 14134.78} C_VEL
LIN {X 0,Y 431.922,Z 1194.239,A -85,B 0,C 180,E1 14132.122,E2 14132.122} C_VEL
LIN {X 0,Y 431.971,Z 1192.507,A -85,B 0,C 180,E1 14129.469,E2 14129.469} C_VEL
LIN {X 0,Y 432.108,Z 1189.73,A -85,B 0,C 180,E1 14126.683,E2 14126.683} C_VEL
LIN {X 0,Y 432.437,Z 1185.911,A -85,B 0,C 180,E1 14123.858,E2 14123.858} C_VEL
LIN {X 0,Y 433.049,Z 1180.95,A -85,B 0,C 180,E1 14120.966,E2 14120.966} C_VEL
LIN {X 0,Y 434.343,Z 1173.636,A -85,B 0,C 180,E1 14117.502,E2 14117.502} C_VEL
LIN {X 0,Y 436.304,Z 1164.491,A -85,B 0,C 180,E1 14114.037,E2 14114.037} C_VEL
LIN {X 0,Y 438.486,Z 1155.858,A -85,B 0,C 180,E1 14111.245,E2 14111.245} C_VEL
LIN {X 0,Y 441.124,Z 1146.488,A -85,B 0,C 180,E1 14108.596,E2 14108.596} C_VEL
LIN {X 0,Y 444.374,Z 1135.914,A -85,B 0,C 180,E1 14105.966,E2 14105.966} C_VEL
LIN {X 0,Y 448.743,Z 1122.51,A -85,B 0,C 180,E1 14103.035,E2 14103.035} C_VEL
LIN {X 0,Y 454.202,Z 1106.394,A -85,B 0,C 180,E1 14100.018,E2 14100.018} C_VEL
LIN {X 0,Y 459.277,Z 1091.689,A -85,B 0,C 180,E1 14097.618,E2 14097.618} C_VEL
LIN {X 0,Y 464.34,Z 1077.103,A -85,B 0,C 180,E1 14095.505,E2 14095.505} C_VEL
LIN {X 0,Y 469.884,Z 1060.968,A -85,B 0,C 180,E1 14093.429,E2 14093.429} C_VEL
LIN {X 0,Y 477.035,Z 1039.633,A -85,B 0,C 180,E1 14091.037,E2 14091.037} C_VEL
LIN {X 0,Y 483.219,Z 1020.185,A -85,B 0,C 180,E1 14089.166,E2 14089.166} C_VEL
LIN {X 0,Y 488.574,Z 1002.626,A -85,B 0,C 180,E1 14087.677,E2 14087.677} C_VEL
LIN {X 0,Y 493.745,Z 984.634,A -85,B 0,C 180,E1 14086.326,E2 14086.326} C_VEL
LIN {X 0,Y 499.136,Z 964.509,A -85,B 0,C 180,E1 14084.997,E2 14084.997} C_VEL
LIN {X 0,Y 505.491,Z 938.455,A -85,B 0,C 180,E1 14083.535,E2 14083.535} C_VEL
LIN {X 0,Y 510.366,Z 915.609,A -85,B 0,C 180,E1 14082.471,E2 14082.471} C_VEL
LIN {X 0,Y 514.229,Z 895.21,A -85,B 0,C 180,E1 14081.666,E2 14081.666} C_VEL
LIN {X 0,Y 517.716,Z 873.969,A -85,B 0,C 180,E1 14080.961,E2 14080.961} C_VEL
LIN {X 0,Y 520.938,Z 850.566,A -85,B 0,C 180,E1 14080.33,E2 14080.33} C_VEL
LIN {X 0,Y 523.932,Z 821.163,A -85,B 0,C 180,E1 14079.738,E2 14079.738} C_VEL
LIN {X 0,Y 527.373,Z 759.317,A -85,B 0,C 180,E1 14078.773,E2 14078.773} C_VEL
LIN {X 0,Y 538.675,Z 547.371,A -85,B 0,C 180,E1 14075.522,E2 14075.522} C_VEL
LIN {X 0,Y 541.863,Z 489.046,A -85,B 0,C 180,E1 14074.615,E2 14074.615} C_VEL
LIN {X 0,Y 534.013,Z 477.064,A -85,B 0,C 180,E1 14072.856,E2 14072.856} C_VEL
LIN {X 0,Y 523.271,Z 461.997,A -85,B 0,C 180,E1 14070.233,E2 14070.233} C_VEL
LIN {X 0,Y 515.223,Z 451.277,A -85,B 0,C 180,E1 14068.043,E2 14068.043} C_VEL
LIN {X 0,Y 508.323,Z 442.17,A -85,B 0,C 180,E1 14065.955,E2 14065.955} C_VEL
LIN {X 0,Y 503.603,Z 436.238,A -85,B 0,C 180,E1 14064.392,E2 14064.392} C_VEL
LIN {X 0,Y 499.648,Z 431.268,A -85,B 0,C 180,E1 14062.969,E2 14062.969} C_VEL
LIN {X 0,Y 495.271,Z 425.881,A -85,B 0,C 180,E1 14061.247,E2 14061.247} C_VEL
LIN {X 0,Y 491.591,Z 421.479,A -85,B 0,C 180,E1 14059.646,E2 14059.646} C_VEL
LIN {X 0,Y 490.558,Z 420.124,A -85,B 0,C 180,E1 14059.157,E2 14059.157} C_VEL
LIN {X 0,Y 487.206,Z 416.542,A -85,B 0,C 180,E1 14057.497,E2 14057.497} C_VEL
LIN {X 0,Y 485.897,Z 414.42,A -85,B 0,C 180,E1 14056.744,E2 14056.744} C_VEL
LIN {X 0,Y 482.308,Z 411.081,A -85,B 0,C 180,E1 14054.589,E2 14054.589} C_VEL
LIN {X 0,Y 480.701,Z 408.096,A -85,B 0,C 180,E1 14053.349,E2 14053.349} C_VEL
LIN {X 0,Y 477.122,Z 405.384,A -85,B 0,C 180,E1 14050.261,E2 14050.261} C_VEL
LIN {X 0,Y 475.556,Z 401.884,A -85,B 0,C 180,E1 14047.977,E2 14047.977} C_VEL
LIN {X 0,Y 473.972,Z 401.215,A -85,B 0,C 180,E1 14042.176,E2 14042.176} C_VEL
LIN {X 0,Y 475.551,Z 401.888,A -85,B 0,C 180,E1 14038.132,E2 14038.132} C_VEL
LIN {X 0,Y 477.268,Z 405.637,A -85,B 0,C 180,E1 14035.675,E2 14035.675} C_VEL
LIN {X 0,Y 480.894,Z 408.501,A -85,B 0,C 180,E1 14032.593,E2 14032.593} C_VEL
LIN {X 0,Y 483.515,Z 412.608,A -85,B 0,C 180,E1 14030.718,E2 14030.718} C_VEL
LIN {X 0,Y 486.15,Z 414.796,A -85,B 0,C 180,E1 14029.213,E2 14029.213} C_VEL
LIN {X 0,Y 489.145,Z 418.914,A -85,B 0,C 180,E1 14027.606,E2 14027.606} C_VEL
LIN {X 0,Y 491.328,Z 421.052,A -85,B 0,C 180,E1 14026.585,E2 14026.585} C_VEL
LIN {X 0,Y 494.736,Z 425.501,A -85,B 0,C 180,E1 14025.067,E2 14025.067} C_VEL
LIN {X 0,Y 496.447,Z 427.407,A -85,B 0,C 180,E1 14024.372,E2 14024.372} C_VEL
LIN {X 0,Y 501.205,Z 433.302,A -85,B 0,C 180,E1 14022.558,E2 14022.558} C_VEL
LIN {X 0,Y 505.879,Z 439.242,A -85,B 0,C 180,E1 14020.936,E2 14020.936} C_VEL
LIN {X 0,Y 510.978,Z 445.723,A -85,B 0,C 180,E1 14019.316,E2 14019.316} C_VEL
LIN {X 0,Y 517.41,Z 454.159,A -85,B 0,C 180,E1 14017.443,E2 14017.443} C_VEL
LIN {X 0,Y 526.935,Z 468.314,A -85,B 0,C 180,E1 14014.906,E2 14014.906} C_VEL
LIN {X 0,Y 536.265,Z 482.808,A -85,B 0,C 180,E1 14012.668,E2 14012.668} C_VEL
LIN {X 0,Y 541.887,Z 491.982,A -85,B 0,C 180,E1 14011.411,E2 14011.411} C_VEL
LIN {X 0,Y 530.377,Z 704.742,A -85,B 0,C 180,E1 14008.141,E2 14008.141} C_VEL
LIN {X 0,Y 523.924,Z 825.479,A -85,B 0,C 180,E1 14006.28,E2 14006.28} C_VEL
LIN {X 0,Y 521.352,Z 852.602,A -85,B 0,C 180,E1 14005.763,E2 14005.763} C_VEL
LIN {X 0,Y 517.705,Z 879.208,A -85,B 0,C 180,E1 14005.072,E2 14005.072} C_VEL
LIN {X 0,Y 514.171,Z 900.669,A -85,B 0,C 180,E1 14004.377,E2 14004.377} C_VEL
LIN {X 0,Y 510.309,Z 921.169,A -85,B 0,C 180,E1 14003.58,E2 14003.58} C_VEL
LIN {X 0,Y 505.835,Z 942.215,A -85,B 0,C 180,E1 14002.62,E2 14002.62} C_VEL
LIN {X 0,Y 499.754,Z 967.929,A -85,B 0,C 180,E1 14001.227,E2 14001.227} C_VEL
LIN {X 0,Y 493.894,Z 989.9,A -85,B 0,C 180,E1 13999.81,E2 13999.81} C_VEL
LIN {X 0,Y 488.531,Z 1008.663,A -85,B 0,C 180,E1 13998.424,E2 13998.424} C_VEL
LIN {X 0,Y 483.084,Z 1026.65,A -85,B 0,C 180,E1 13996.918,E2 13996.918} C_VEL
LIN {X 0,Y 477.068,Z 1045.72,A -85,B 0,C 180,E1 13995.106,E2 13995.106} C_VEL
LIN {X 0,Y 469.636,Z 1068.272,A -85,B 0,C 180,E1 13992.613,E2 13992.613} C_VEL
LIN {X 0,Y 464.209,Z 1084.251,A -85,B 0,C 180,E1 13990.579,E2 13990.579} C_VEL
LIN {X 0,Y 459.271,Z 1098.72,A -85,B 0,C 180,E1 13988.51,E2 13988.51} C_VEL
LIN {X 0,Y 454.533,Z 1112.632,A -85,B 0,C 180,E1 13986.281,E2 13986.281} C_VEL
LIN {X 0,Y 449.621,Z 1127.33,A -85,B 0,C 180,E1 13983.624,E2 13983.624} C_VEL
LIN {X 0,Y 444.504,Z 1143.313,A -85,B 0,C 180,E1 13980.255,E2 13980.255} C_VEL
LIN {X 0,Y 441.139,Z 1154.452,A -85,B 0,C 180,E1 13977.541,E2 13977.541} C_VEL
LIN {X 0,Y 438.429,Z 1164.296,A -85,B 0,C 180,E1 13974.812,E2 13974.812} C_VEL
LIN {X 0,Y 436.206,Z 1173.328,A -85,B 0,C 180,E1 13971.94,E2 13971.94} C_VEL
LIN {X 0,Y 434.221,Z 1182.823,A -85,B 0,C 180,E1 13968.39,E2 13968.39} C_VEL
LIN {X 0,Y 433.018,Z 1190.12,A -85,B 0,C 180,E1 13964.989,E2 13964.989} C_VEL
LIN {X 0,Y 432.412,Z 1195.096,A -85,B 0,C 180,E1 13962.148,E2 13962.148} C_VEL
LIN {X 0,Y 432.104,Z 1198.846,A -85,B 0,C 180,E1 13959.457,E2 13959.457} C_VEL
LIN {X 0,Y 431.965,Z 1201.661,A -85,B 0,C 180,E1 13956.767,E2 13956.767} C_VEL
LIN {X 0,Y 431.917,Z 1203.525,A -85,B 0,C 180,E1 13954.116,E2 13954.116} C_VEL
LIN {X 0,Y 431.912,Z 1204.483,A -85,B 0,C 180,E1 13951.46,E2 13951.46} C_VEL
LIN {X 0,Y 431.913,Z 1204.528,A -85,B 0,C 180,E1 13948.807,E2 13948.807} C_VEL
LIN {X 0,Y 431.914,Z 1203.659,A -85,B 0,C 180,E1 13946.151,E2 13946.151} C_VEL
LIN {X 0,Y 431.959,Z 1201.874,A -85,B 0,C 180,E1 13943.488,E2 13943.488} C_VEL
LIN {X 0,Y 432.084,Z 1199.161,A -85,B 0,C 180,E1 13940.813,E2 13940.813} C_VEL
LIN {X 0,Y 432.367,Z 1195.503,A -85,B 0,C 180,E1 13938.123,E2 13938.123} C_VEL
LIN {X 0,Y 432.915,Z 1190.86,A -85,B 0,C 180,E1 13935.411,E2 13935.411} C_VEL
LIN {X 0,Y 433.808,Z 1185.021,A -85,B 0,C 180,E1 13932.6,E2 13932.6} C_VEL
LIN {X 0,Y 435.27,Z 1177.519,A -85,B 0,C 180,E1 13929.564,E2 13929.564} C_VEL
LIN {X 0,Y 437.96,Z 1166.155,A -85,B 0,C 180,E1 13925.736,E2 13925.736} C_VEL
LIN {X 0,Y 440.849,Z 1155.592,A -85,B 0,C 180,E1 13922.733,E2 13922.733} C_VEL
LIN {X 0,Y 444.164,Z 1144.713,A -85,B 0,C 180,E1 13920.017,E2 13920.017} C_VEL
LIN {X 0,Y 448.352,Z 1131.871,A -85,B 0,C 180,E1 13917.186,E2 13917.186} C_VEL
LIN {X 0,Y 454.438,Z 1114.292,A -85,B 0,C 180,E1 13913.853,E2 13913.853} C_VEL
LIN {X 0,Y 459.783,Z 1099.259,A -85,B 0,C 180,E1 13911.382,E2 13911.382} C_VEL
LIN {X 0,Y 465.166,Z 1084.287,A -85,B 0,C 180,E1 13909.199,E2 13909.199} C_VEL
LIN {X 0,Y 471.481,Z 1066.733,A -85,B 0,C 180,E1 13906.933,E2 13906.933} C_VEL
LIN {X 0,Y 479.204,Z 1044.57,A -85,B 0,C 180,E1 13904.473,E2 13904.473} C_VEL
LIN {X 0,Y 485.3,Z 1026.487,A -85,B 0,C 180,E1 13902.735,E2 13902.735} C_VEL
LIN {X 0,Y 491.119,Z 1008.51,A -85,B 0,C 180,E1 13901.214,E2 13901.214} C_VEL
LIN {X 0,Y 496.774,Z 990.094,A -85,B 0,C 180,E1 13899.839,E2 13899.839} C_VEL
LIN {X 0,Y 502.942,Z 968.604,A -85,B 0,C 180,E1 13898.438,E2 13898.438} C_VEL
LIN {X 0,Y 509.61,Z 942.548,A -85,B 0,C 180,E1 13897.009,E2 13897.009} C_VEL
LIN {X 0,Y 514.428,Z 921.551,A -85,B 0,C 180,E1 13896.045,E2 13896.045} C_VEL
LIN {X 0,Y 518.547,Z 901.342,A -85,B 0,C 180,E1 13895.255,E2 13895.255} C_VEL
LIN {X 0,Y 522.434,Z 879.531,A -85,B 0,C 180,E1 13894.546,E2 13894.546} C_VEL
LIN {X 0,Y 526.149,Z 854.57,A -85,B 0,C 180,E1 13893.892,E2 13893.892} C_VEL
LIN {X 0,Y 529.149,Z 826.391,A -85,B 0,C 180,E1 13893.343,E2 13893.343} C_VEL
LIN {X 0,Y 534.278,Z 742.415,A -85,B 0,C 180,E1 13892.025,E2 13892.025} C_VEL
LIN {X 0,Y 547.597,Z 524.77,A -85,B 0,C 180,E1 13888.645,E2 13888.645} C_VEL
LIN {X 0,Y 549.444,Z 494.333,A -85,B 0,C 180,E1 13888.151,E2 13888.151} C_VEL
LIN {X 0,Y 541.295,Z 481.078,A -85,B 0,C 180,E1 13885.875,E2 13885.875} C_VEL
LIN {X 0,Y 532.442,Z 467.899,A -85,B 0,C 180,E1 13883.08,E2 13883.08} C_VEL
LIN {X 0,Y 527.574,Z 461.035,A -85,B 0,C 180,E1 13881.339,E2 13881.339} C_VEL
LIN {X 0,Y 524.849,Z 457.438,A -85,B 0,C 180,E1 13880.287,E2 13880.287} C_VEL
LIN {X 0,Y 521.058,Z 452.482,A -85,B 0,C 180,E1 13878.691,E2 13878.691} C_VEL
LIN {X 0,Y 516.98,Z 447.21,A -85,B 0,C 180,E1 13876.749,E2 13876.749} C_VEL
LIN {X 0,Y 513.424,Z 442.757,A -85,B 0,C 180,E1 13874.781,E2 13874.781} C_VEL
LIN {X 0,Y 512.535,Z 441.605,A -85,B 0,C 180,E1 13874.23,E2 13874.23} C_VEL
LIN {X 0,Y 509.479,Z 438.291,A -85,B 0,C 180,E1 13872.122,E2 13872.122} C_VEL
LIN {X 0,Y 508.105,Z 435.771,A -85,B 0,C 180,E1 13870.89,E2 13870.89} C_VEL
LIN {X 0,Y 504.749,Z 432.695,A -85,B 0,C 180,E1 13866.941,E2 13866.941} C_VEL
LIN {X 0,Y 503.871,Z 429.607,A -85,B 0,C 180,E1 13863.499,E2 13863.499} C_VEL
LIN {X 0,Y 503.904,Z 429.871,A -85,B 0,C 180,E1 13861.819,E2 13861.819} C_VEL
LIN {X 0,Y 506.865,Z 435.024,A -85,B 0,C 180,E1 13856.041,E2 13856.041} C_VEL
LIN {X 0,Y 508.4,Z 436.164,A -85,B 0,C 180,E1 13854.64,E2 13854.64} C_VEL
LIN {X 0,Y 510.79,Z 440.003,A -85,B 0,C 180,E1 13852.69,E2 13852.69} C_VEL
LIN {X 0,Y 513.219,Z 442.384,A -85,B 0,C 180,E1 13851.146,E2 13851.146} C_VEL
LIN {X 0,Y 516.276,Z 446.555,A -85,B 0,C 180,E1 13849.398,E2 13849.398} C_VEL
LIN {X 0,Y 517.907,Z 448.281,A -85,B 0,C 180,E1 13848.586,E2 13848.586} C_VEL
LIN {X 0,Y 522.583,Z 454.385,A -85,B 0,C 180,E1 13846.444,E2 13846.444} C_VEL
LIN {X 0,Y 526.924,Z 460.045,A -85,B 0,C 180,E1 13844.706,E2 13844.706} C_VEL
LIN {X 0,Y 531.374,Z 465.94,A -85,B 0,C 180,E1 13843.099,E2 13843.099} C_VEL
LIN {X 0,Y 537.639,Z 474.449,A -85,B 0,C 180,E1 13841.063,E2 13841.063} C_VEL
LIN {X 0,Y 546.43,Z 486.913,A -85,B 0,C 180,E1 13838.532,E2 13838.532} C_VEL
LIN {X 0,Y 549.547,Z 491.936,A -85,B 0,C 180,E1 13837.693,E2 13837.693} C_VEL
LIN {X 0,Y 536.405,Z 703.813,A -85,B 0,C 180,E1 13834.401,E2 13834.401} C_VEL
LIN {X 0,Y 529.386,Z 819.484,A -85,B 0,C 180,E1 13832.593,E2 13832.593} C_VEL
LIN {X 0,Y 526.576,Z 846.815,A -85,B 0,C 180,E1 13832.065,E2 13832.065} C_VEL
LIN {X 0,Y 522.716,Z 873.072,A -85,B 0,C 180,E1 13831.372,E2 13831.372} C_VEL
LIN {X 0,Y 518.982,Z 894.253,A -85,B 0,C 180,E1 13830.678,E2 13830.678} C_VEL
LIN {X 0,Y 514.928,Z 914.335,A -85,B 0,C 180,E1 13829.889,E2 13829.889} C_VEL
LIN {X 0,Y 510.151,Z 935.264,A -85,B 0,C 180,E1 13828.925,E2 13828.925} C_VEL
LIN {X 0,Y 503.957,Z 959.822,A -85,B 0,C 180,E1 13827.587,E2 13827.587} C_VEL
LIN {X 0,Y 497.447,Z 982.475,A -85,B 0,C 180,E1 13826.112,E2 13826.112} C_VEL
LIN {X 0,Y 491.755,Z 1000.975,A -85,B 0,C 180,E1 13824.728,E2 13824.728} C_VEL
LIN {X 0,Y 485.842,Z 1019.145,A -85,B 0,C 180,E1 13823.184,E2 13823.184} C_VEL
LIN {X 0,Y 479.63,Z 1037.402,A -85,B 0,C 180,E1 13821.421,E2 13821.421} C_VEL
LIN {X 0,Y 471.898,Z 1059.365,A -85,B 0,C 180,E1 13818.964,E2 13818.964} C_VEL
LIN {X 0,Y 465.589,Z 1076.63,A -85,B 0,C 180,E1 13816.72,E2 13816.72} C_VEL
LIN {X 0,Y 460.172,Z 1091.428,A -85,B 0,C 180,E1 13814.545,E2 13814.545} C_VEL
LIN {X 0,Y 455.111,Z 1105.396,A -85,B 0,C 180,E1 13812.234,E2 13812.234} C_VEL
LIN {X 0,Y 449.403,Z 1121.614,A -85,B 0,C 180,E1 13809.187,E2 13809.187} C_VEL
LIN {X 0,Y 444.648,Z 1135.613,A -85,B 0,C 180,E1 13806.096,E2 13806.096} C_VEL
LIN {X 0,Y 441.271,Z 1146.32,A -85,B 0,C 180,E1 13803.408,E2 13803.408} C_VEL
LIN {X 0,Y 438.543,Z 1155.793,A -85,B 0,C 180,E1 13800.711,E2 13800.711} C_VEL
LIN {X 0,Y 436.12,Z 1165.361,A -85,B 0,C 180,E1 13797.588,E2 13797.588} C_VEL
LIN {X 0,Y 434.055,Z 1175.056,A -85,B 0,C 180,E1 13793.773,E2 13793.773} C_VEL
LIN {X 0,Y 433.028,Z 1181.177,A -85,B 0,C 180,E1 13790.829,E2 13790.829} C_VEL
LIN {X 0,Y 432.575,Z 1184.656,A -85,B 0,C 180,E1 13788.889,E2 13788.889} C_VEL
LIN {X 0,Y 431.414,Z 1186.254,A -85,B 0,C 180,E1 13787.891,E2 13787.891} C_VEL
LIN {X 0,Y 424.75,Z 1190.119,A -85,B 0,C 180,E1 13785.154,E2 13785.154} C_VEL
LIN {X 0,Y 424.054,Z 1191.052,A -85,B 0,C 180,E1 13784.342,E2 13784.342} C_VEL
LIN {X 0,Y 423.928,Z 1193.894,A -85,B 0,C 180,E1 13780.738,E2 13780.738} C_VEL
LIN {X 0,Y 423.912,Z 1195.076,A -85,B 0,C 180,E1 13777.726,E2 13777.726} C_VEL
LIN {X 0,Y 423.904,Z 1195.212,A -85,B 0,C 180,E1 13775.006,E2 13775.006} C_VEL
LIN {X 0,Y 423.922,Z 1194.382,A -85,B 0,C 180,E1 13772.162,E2 13772.162} C_VEL
LIN {X 0,Y 423.973,Z 1192.687,A -85,B 0,C 180,E1 13769.459,E2 13769.459} C_VEL
LIN {X 0,Y 424.117,Z 1189.947,A -85,B 0,C 180,E1 13766.621,E2 13766.621} C_VEL
LIN {X 0,Y 424.458,Z 1186.217,A -85,B 0,C 180,E1 13763.776,E2 13763.776} C_VEL
LIN {X 0,Y 425.07,Z 1181.493,A -85,B 0,C 180,E1 13760.932,E2 13760.932} C_VEL
LIN {X 0,Y 426.093,Z 1175.736,A -85,B 0,C 180,E1 13758.082,E2 13758.082} C_VEL
LIN {X 0,Y 427.796,Z 1167.885,A -85,B 0,C 180,E1 13754.824,E2 13754.824} C_VEL
LIN {X 0,Y 430.571,Z 1157.172,A -85,B 0,C 180,E1 13751.168,E2 13751.168} C_VEL
LIN {X 0,Y 433.576,Z 1146.937,A -85,B 0,C 180,E1 13748.205,E2 13748.205} C_VEL
LIN {X 0,Y 436.966,Z 1136.388,A -85,B 0,C 180,E1 13745.533,E2 13745.533} C_VEL
LIN {X 0,Y 441.177,Z 1123.933,A -85,B 0,C 180,E1 13742.754,E2 13742.754} C_VEL
LIN {X 0,Y 447.192,Z 1106.964,A -85,B 0,C 180,E1 13739.499,E2 13739.499} C_VEL
LIN {X 0,Y 452.447,Z 1092.292,A -85,B 0,C 180,E1 13737.068,E2 13737.068} C_VEL
LIN {X 0,Y 457.692,Z 1077.743,A -85,B 0,C 180,E1 13734.931,E2 13734.931} C_VEL
LIN {X 0,Y 463.07,Z 1062.632,A -85,B 0,C 180,E1 13732.956,E2 13732.956} C_VEL
LIN {X 0,Y 469.282,Z 1044.857,A -85,B 0,C 180,E1 13730.9,E2 13730.9} C_VEL
LIN {X 0,Y 476.779,Z 1022.321,A -85,B 0,C 180,E1 13728.654,E2 13728.654} C_VEL
LIN {X 0,Y 482.695,Z 1003.522,A -85,B 0,C 180,E1 13727.038,E2 13727.038} C_VEL
LIN {X 0,Y 488.017,Z 985.605,A -85,B 0,C 180,E1 13725.68,E2 13725.68} C_VEL
LIN {X 0,Y 493.314,Z 966.447,A -85,B 0,C 180,E1 13724.4,E2 13724.4} C_VEL
LIN {X 0,Y 499.115,Z 943.746,A -85,B 0,C 180,E1 13723.089,E2 13723.089} C_VEL
LIN {X 0,Y 504.83,Z 918.293,A -85,B 0,C 180,E1 13721.865,E2 13721.865} C_VEL
LIN {X 0,Y 509.089,Z 896.584,A -85,B 0,C 180,E1 13720.996,E2 13720.996} C_VEL
LIN {X 0,Y 512.693,Z 875.335,A -85,B 0,C 180,E1 13720.283,E2 13720.283} C_VEL
LIN {X 0,Y 515.78,Z 853.76,A -85,B 0,C 180,E1 13719.691,E2 13719.691} C_VEL
LIN {X 0,Y 518.809,Z 827.279,A -85,B 0,C 180,E1 13719.124,E2 13719.124} C_VEL
LIN {X 0,Y 521.416,Z 785.511,A -85,B 0,C 180,E1 13718.454,E2 13718.454} C_VEL
LIN {X 0,Y 533.433,Z 566.149,A -85,B 0,C 180,E1 13715.082,E2 13715.082} C_VEL
LIN {X 0,Y 537.548,Z 493.429,A -85,B 0,C 180,E1 13713.952,E2 13713.952} C_VEL
LIN {X 0,Y 529.67,Z 481.636,A -85,B 0,C 180,E1 13712.133,E2 13712.133} C_VEL
LIN {X 0,Y 520.454,Z 468.525,A -85,B 0,C 180,E1 13709.809,E2 13709.809} C_VEL
LIN {X 0,Y 512.724,Z 458.086,A -85,B 0,C 180,E1 13707.655,E2 13707.655} C_VEL
LIN {X 0,Y 506.024,Z 449.171,A -85,B 0,C 180,E1 13705.579,E2 13705.579} C_VEL
LIN {X 0,Y 501.547,Z 443.445,A -85,B 0,C 180,E1 13704.06,E2 13704.06} C_VEL
LIN {X 0,Y 497.806,Z 438.679,A -85,B 0,C 180,E1 13702.684,E2 13702.684} C_VEL
LIN {X 0,Y 493.498,Z 433.334,A -85,B 0,C 180,E1 13700.954,E2 13700.954} C_VEL
LIN {X 0,Y 489.83,Z 428.747,A -85,B 0,C 180,E1 13699.311,E2 13699.311} C_VEL
LIN {X 0,Y 485.405,Z 423.608,A -85,B 0,C 180,E1 13697.07,E2 13697.07} C_VEL
LIN {X 0,Y 484.518,Z 422.177,A -85,B 0,C 180,E1 13696.546,E2 13696.546} C_VEL
LIN {X 0,Y 480.916,Z 418.66,A -85,B 0,C 180,E1 13694.325,E2 13694.325} C_VEL
LIN {X 0,Y 479.414,Z 415.919,A -85,B 0,C 180,E1 13693.14,E2 13693.14} C_VEL
LIN {X 0,Y 475.94,Z 413.12,A -85,B 0,C 180,E1 13690.042,E2 13690.042} C_VEL
LIN {X 0,Y 474.367,Z 409.623,A -85,B 0,C 180,E1 13687.631,E2 13687.631} C_VEL
LIN {X 0,Y 473.139,Z 409.235,A -85,B 0,C 180,E1 13681.332,E2 13681.332} C_VEL
LIN {X 0,Y 474.495,Z 409.797,A -85,B 0,C 180,E1 13678.249,E2 13678.249} C_VEL
LIN {X 0,Y 476.286,Z 413.64,A -85,B 0,C 180,E1 13675.666,E2 13675.666} C_VEL
LIN {X 0,Y 479.669,Z 416.349,A -85,B 0,C 180,E1 13672.755,E2 13672.755} C_VEL
LIN {X 0,Y 482.347,Z 420.494,A -85,B 0,C 180,E1 13670.815,E2 13670.815} C_VEL
LIN {X 0,Y 484.844,Z 422.69,A -85,B 0,C 180,E1 13669.364,E2 13669.364} C_VEL
LIN {X 0,Y 487.932,Z 426.819,A -85,B 0,C 180,E1 13667.695,E2 13667.695} C_VEL
LIN {X 0,Y 489.732,Z 428.593,A -85,B 0,C 180,E1 13666.841,E2 13666.841} C_VEL
LIN {X 0,Y 493.217,Z 433.177,A -85,B 0,C 180,E1 13665.26,E2 13665.26} C_VEL
LIN {X 0,Y 494.834,Z 435.056,A -85,B 0,C 180,E1 13664.59,E2 13664.59} C_VEL
LIN {X 0,Y 499.532,Z 440.966,A -85,B 0,C 180,E1 13662.768,E2 13662.768} C_VEL
LIN {X 0,Y 504.075,Z 446.812,A -85,B 0,C 180,E1 13661.166,E2 13661.166} C_VEL
LIN {X 0,Y 509.035,Z 453.181,A -85,B 0,C 180,E1 13659.564,E2 13659.564} C_VEL
LIN {X 0,Y 515.571,Z 461.941,A -85,B 0,C 180,E1 13657.629,E2 13657.629} C_VEL
LIN {X 0,Y 526.003,Z 477.721,A -85,B 0,C 180,E1 13654.828,E2 13654.828} C_VEL
LIN {X 0,Y 535.953,Z 493.658,A -85,B 0,C 180,E1 13652.44,E2 13652.44} C_VEL
LIN {X 0,Y 537.532,Z 496.524,A -85,B 0,C 180,E1 13652.075,E2 13652.075} C_VEL
LIN {X 0,Y 525.61,Z 710.295,A -85,B 0,C 180,E1 13648.78,E2 13648.78} C_VEL
LIN {X 0,Y 519.241,Z 825.549,A -85,B 0,C 180,E1 13646.995,E2 13646.995} C_VEL
LIN {X 0,Y 516.581,Z 852.865,A -85,B 0,C 180,E1 13646.473,E2 13646.473} C_VEL
LIN {X 0,Y 512.844,Z 879.383,A -85,B 0,C 180,E1 13645.782,E2 13645.782} C_VEL
LIN {X 0,Y 509.289,Z 900.435,A -85,B 0,C 180,E1 13645.101,E2 13645.101} C_VEL
LIN {X 0,Y 505.354,Z 920.792,A -85,B 0,C 180,E1 13644.312,E2 13644.312} C_VEL
LIN {X 0,Y 500.856,Z 941.436,A -85,B 0,C 180,E1 13643.373,E2 13643.373} C_VEL
LIN {X 0,Y 495.023,Z 965.738,A -85,B 0,C 180,E1 13642.07,E2 13642.07} C_VEL
LIN {X 0,Y 488.636,Z 989.057,A -85,B 0,C 180,E1 13640.576,E2 13640.576} C_VEL
LIN {X 0,Y 482.993,Z 1008.221,A -85,B 0,C 180,E1 13639.161,E2 13639.161} C_VEL
LIN {X 0,Y 477.442,Z 1026.017,A -85,B 0,C 180,E1 13637.669,E2 13637.669} C_VEL
LIN {X 0,Y 471.446,Z 1044.408,A -85,B 0,C 180,E1 13635.92,E2 13635.92} C_VEL
LIN {X 0,Y 464.195,Z 1065.848,A -85,B 0,C 180,E1 13633.574,E2 13633.574} C_VEL
LIN {X 0,Y 457.826,Z 1083.927,A -85,B 0,C 180,E1 13631.267,E2 13631.267} C_VEL
LIN {X 0,Y 452.65,Z 1098.518,A -85,B 0,C 180,E1 13629.163,E2 13629.163} C_VEL
LIN {X 0,Y 447.729,Z 1112.398,A -85,B 0,C 180,E1 13626.917,E2 13626.917} C_VEL
LIN {X 0,Y 442.869,Z 1126.386,A -85,B 0,C 180,E1 13624.363,E2 13624.363} C_VEL
LIN {X 0,Y 437.428,Z 1142.533,A -85,B 0,C 180,E1 13620.952,E2 13620.952} C_VEL
LIN {X 0,Y 433.712,Z 1154.289,A -85,B 0,C 180,E1 13618.054,E2 13618.054} C_VEL
LIN {X 0,Y 430.974,Z 1163.693,A -85,B 0,C 180,E1 13615.418,E2 13615.418} C_VEL
LIN {X 0,Y 428.675,Z 1172.396,A -85,B 0,C 180,E1 13612.635,E2 13612.635} C_VEL
LIN {X 0,Y 426.854,Z 1180.423,A -85,B 0,C 180,E1 13609.665,E2 13609.665} C_VEL
LIN {X 0,Y 425.272,Z 1189.003,A -85,B 0,C 180,E1 13605.827,E2 13605.827} C_VEL
LIN {X 0,Y 424.493,Z 1194.59,A -85,B 0,C 180,E1 13602.654,E2 13602.654} C_VEL
LIN {X 0,Y 424.134,Z 1198.596,A -85,B 0,C 180,E1 13599.773,E2 13599.773} C_VEL
LIN {X 0,Y 423.973,Z 1201.447,A -85,B 0,C 180,E1 13597.045,E2 13597.045} C_VEL
LIN {X 0,Y 423.918,Z 1203.369,A -85,B 0,C 180,E1 13594.329,E2 13594.329} C_VEL
LIN {X 0,Y 423.91,Z 1204.373,A -85,B 0,C 180,E1 13591.622,E2 13591.622} C_VEL
LIN {X 0,Y 423.911,Z 1204.463,A -85,B 0,C 180,E1 13588.919,E2 13588.919} C_VEL
LIN {X 0,Y 423.915,Z 1203.64,A -85,B 0,C 180,E1 13586.214,E2 13586.214} C_VEL
LIN {X 0,Y 423.959,Z 1201.899,A -85,B 0,C 180,E1 13583.5,E2 13583.5} C_VEL
LIN {X 0,Y 424.087,Z 1199.232,A -85,B 0,C 180,E1 13580.775,E2 13580.775} C_VEL
LIN {X 0,Y 424.383,Z 1195.621,A -85,B 0,C 180,E1 13578.034,E2 13578.034} C_VEL
LIN {X 0,Y 424.986,Z 1190.783,A -85,B 0,C 180,E1 13575.141,E2 13575.141} C_VEL
LIN {X 0,Y 425.958,Z 1184.851,A -85,B 0,C 180,E1 13572.233,E2 13572.233} C_VEL
LIN {X 0,Y 427.583,Z 1177.084,A -85,B 0,C 180,E1 13569.037,E2 13569.037} C_VEL
LIN {X 0,Y 430.482,Z 1165.652,A -85,B 0,C 180,E1 13565.14,E2 13565.14} C_VEL
LIN {X 0,Y 433.42,Z 1155.576,A -85,B 0,C 180,E1 13562.226,E2 13562.226} C_VEL
LIN {X 0,Y 436.92,Z 1144.723,A -85,B 0,C 180,E1 13559.467,E2 13559.467} C_VEL
LIN {X 0,Y 441.082,Z 1132.543,A -85,B 0,C 180,E1 13556.731,E2 13556.731} C_VEL
LIN {X 0,Y 447.395,Z 1115.214,A -85,B 0,C 180,E1 13553.366,E2 13553.366} C_VEL
LIN {X 0,Y 452.961,Z 1100.214,A -85,B 0,C 180,E1 13550.853,E2 13550.853} C_VEL
LIN {X 0,Y 458.535,Z 1085.356,A -85,B 0,C 180,E1 13548.646,E2 13548.646} C_VEL
LIN {X 0,Y 464.306,Z 1069.925,A -85,B 0,C 180,E1 13546.611,E2 13546.611} C_VEL
LIN {X 0,Y 470.991,Z 1051.792,A -85,B 0,C 180,E1 13544.497,E2 13544.497} C_VEL
LIN {X 0,Y 479.096,Z 1028.754,A -85,B 0,C 180,E1 13542.194,E2 13542.194} C_VEL
LIN {X 0,Y 485.18,Z 1010.677,A -85,B 0,C 180,E1 13540.635,E2 13540.635} C_VEL
LIN {X 0,Y 490.861,Z 992.883,A -85,B 0,C 180,E1 13539.282,E2 13539.282} C_VEL
LIN {X 0,Y 496.381,Z 974.377,A -85,B 0,C 180,E1 13538.039,E2 13538.039} C_VEL
LIN {X 0,Y 502.126,Z 953.576,A -85,B 0,C 180,E1 13536.823,E2 13536.823} C_VEL
LIN {X 0,Y 508.39,Z 928.564,A -85,B 0,C 180,E1 13535.586,E2 13535.586} C_VEL
LIN {X 0,Y 513.705,Z 903.611,A -85,B 0,C 180,E1 13534.582,E2 13534.582} C_VEL
LIN {X 0,Y 517.662,Z 882.326,A -85,B 0,C 180,E1 13533.876,E2 13533.876} C_VEL
LIN {X 0,Y 520.959,Z 861.3,A -85,B 0,C 180,E1 13533.303,E2 13533.303} C_VEL
LIN {X 0,Y 523.917,Z 838.075,A -85,B 0,C 180,E1 13532.803,E2 13532.803} C_VEL
LIN {X 0,Y 526.727,Z 802.169,A -85,B 0,C 180,E1 13532.199,E2 13532.199} C_VEL
LIN {X 0,Y 540.454,Z 580.626,A -85,B 0,C 180,E1 13528.757,E2 13528.757} C_VEL
LIN {X 0,Y 545.704,Z 499.04,A -85,B 0,C 180,E1 13527.47,E2 13527.47} C_VEL
LIN {X 0,Y 538.105,Z 486.758,A -85,B 0,C 180,E1 13525.272,E2 13525.272} C_VEL
LIN {X 0,Y 529.323,Z 473.277,A -85,B 0,C 180,E1 13522.373,E2 13522.373} C_VEL
LIN {X 0,Y 523.486,Z 465.293,A -85,B 0,C 180,E1 13520.168,E2 13520.168} C_VEL
LIN {X 0,Y 519.364,Z 459.931,A -85,B 0,C 180,E1 13518.405,E2 13518.405} C_VEL
LIN {X 0,Y 515.586,Z 454.92,A -85,B 0,C 180,E1 13516.564,E2 13516.564} C_VEL
LIN {X 0,Y 512.005,Z 450.313,A -85,B 0,C 180,E1 13514.534,E2 13514.534} C_VEL
LIN {X 0,Y 511.032,Z 449.227,A -85,B 0,C 180,E1 13513.926,E2 13513.926} C_VEL
LIN {X 0,Y 508.099,Z 445.756,A -85,B 0,C 180,E1 13511.81,E2 13511.81} C_VEL
LIN {X 0,Y 507.01,Z 443.669,A -85,B 0,C 180,E1 13510.798,E2 13510.798} C_VEL
LIN {X 0,Y 503.714,Z 440.579,A -85,B 0,C 180,E1 13506.84,E2 13506.84} C_VEL
LIN {X 0,Y 502.887,Z 437.552,A -85,B 0,C 180,E1 13503.42,E2 13503.42} C_VEL
LIN {X 0,Y 502.921,Z 437.857,A -85,B 0,C 180,E1 13501.823,E2 13501.823} C_VEL
LIN {X 0,Y 505.887,Z 442.985,A -85,B 0,C 180,E1 13496.033,E2 13496.033} C_VEL
LIN {X 0,Y 507.224,Z 443.978,A -85,B 0,C 180,E1 13494.797,E2 13494.797} C_VEL
LIN {X 0,Y 509.648,Z 447.881,A -85,B 0,C 180,E1 13492.787,E2 13492.787} C_VEL
LIN {X 0,Y 511.872,Z 450.068,A -85,B 0,C 180,E1 13491.349,E2 13491.349} C_VEL
LIN {X 0,Y 515.084,Z 454.443,A -85,B 0,C 180,E1 13489.486,E2 13489.486} C_VEL
LIN {X 0,Y 516.58,Z 456.152,A -85,B 0,C 180,E1 13488.726,E2 13488.726} C_VEL
LIN {X 0,Y 520.964,Z 461.915,A -85,B 0,C 180,E1 13486.684,E2 13486.684} C_VEL
LIN {X 0,Y 525.505,Z 467.969,A -85,B 0,C 180,E1 13484.833,E2 13484.833} C_VEL
LIN {X 0,Y 529.921,Z 473.888,A -85,B 0,C 180,E1 13483.22,E2 13483.22} C_VEL
LIN {X 0,Y 536.291,Z 482.761,A -85,B 0,C 180,E1 13481.126,E2 13481.126} C_VEL
LIN {X 0,Y 544.319,Z 494.333,A -85,B 0,C 180,E1 13478.784,E2 13478.784} C_VEL
LIN {X 0,Y 545.767,Z 496.903,A -85,B 0,C 180,E1 13478.377,E2 13478.377} C_VEL
LIN {X 0,Y 532.317,Z 707.341,A -85,B 0,C 180,E1 13475.101,E2 13475.101} C_VEL
LIN {X 0,Y 525.286,Z 819.576,A -85,B 0,C 180,E1 13473.343,E2 13473.343} C_VEL
LIN {X 0,Y 522.398,Z 846.973,A -85,B 0,C 180,E1 13472.814,E2 13472.814} C_VEL
LIN {X 0,Y 518.463,Z 873.081,A -85,B 0,C 180,E1 13472.127,E2 13472.127} C_VEL
LIN {X 0,Y 514.599,Z 894.407,A -85,B 0,C 180,E1 13471.43,E2 13471.43} C_VEL
LIN {X 0,Y 510.322,Z 915.003,A -85,B 0,C 180,E1 13470.621,E2 13470.621} C_VEL
LIN {X 0,Y 505.277,Z 936.443,A -85,B 0,C 180,E1 13469.63,E2 13469.63} C_VEL
LIN {X 0,Y 498.321,Z 962.709,A -85,B 0,C 180,E1 13468.172,E2 13468.172} C_VEL
LIN {X 0,Y 492.214,Z 983.314,A -85,B 0,C 180,E1 13466.816,E2 13466.816} C_VEL
LIN {X 0,Y 486.582,Z 1001.025,A -85,B 0,C 180,E1 13465.487,E2 13465.487} C_VEL
LIN {X 0,Y 480.488,Z 1019.138,A -85,B 0,C 180,E1 13463.944,E2 13463.944} C_VEL
LIN {X 0,Y 474.056,Z 1037.398,A -85,B 0,C 180,E1 13462.174,E2 13462.174} C_VEL
LIN {X 0,Y 466.026,Z 1059.355,A -85,B 0,C 180,E1 13459.705,E2 13459.705} C_VEL
LIN {X 0,Y 459.651,Z 1076.145,A -85,B 0,C 180,E1 13457.512,E2 13457.512} C_VEL
LIN {X 0,Y 454.036,Z 1090.84,A -85,B 0,C 180,E1 13455.341,E2 13455.341} C_VEL
LIN {X 0,Y 448.682,Z 1104.946,A -85,B 0,C 180,E1 13452.992,E2 13452.992} C_VEL
LIN {X 0,Y 442.908,Z 1120.548,A -85,B 0,C 180,E1 13450.045,E2 13450.045} C_VEL
LIN {X 0,Y 437.617,Z 1135.302,A -85,B 0,C 180,E1 13446.771,E2 13446.771} C_VEL
LIN {X 0,Y 433.914,Z 1146.388,A -85,B 0,C 180,E1 13443.945,E2 13443.945} C_VEL
LIN {X 0,Y 430.937,Z 1156.155,A -85,B 0,C 180,E1 13441.109,E2 13441.109} C_VEL
LIN {X 0,Y 428.119,Z 1166.783,A -85,B 0,C 180,E1 13437.543,E2 13437.543} C_VEL
LIN {X 0,Y 426.144,Z 1175.503,A -85,B 0,C 180,E1 13433.948,E2 13433.948} C_VEL
LIN {X 0,Y 425.116,Z 1181.305,A -85,B 0,C 180,E1 13431.091,E2 13431.091} C_VEL
LIN {X 0,Y 424.482,Z 1186.048,A -85,B 0,C 180,E1 13428.257,E2 13428.257} C_VEL
LIN {X 0,Y 424.131,Z 1189.771,A -85,B 0,C 180,E1 13425.449,E2 13425.449} C_VEL
LIN {X 0,Y 424.054,Z 1191.052,A -85,B 0,C 180,E1 13424.342,E2 13424.342} C_VEL
LIN {X 0,Y 423.001,Z 1192.131,A -85,B 0,C 180,E1 13423.312,E2 13423.312} C_VEL
LIN {X 0,Y 416.452,Z 1194.191,A -85,B 0,C 180,E1 13420.397,E2 13420.397} C_VEL
LIN {X 0,Y 415.919,Z 1194.564,A -85,B 0,C 180,E1 13419.633,E2 13419.633} C_VEL
LIN {X 0,Y 415.9,Z 1195.37,A -85,B 0,C 180,E1 13416.487,E2 13416.487} C_VEL
LIN {X 0,Y 415.915,Z 1194.862,A -85,B 0,C 180,E1 13412.893,E2 13412.893} C_VEL
LIN {X 0,Y 415.971,Z 1192.978,A -85,B 0,C 180,E1 13409.586,E2 13409.586} C_VEL
LIN {X 0,Y 416.127,Z 1190.165,A -85,B 0,C 180,E1 13406.556,E2 13406.556} C_VEL
LIN {X 0,Y 416.485,Z 1186.477,A -85,B 0,C 180,E1 13403.659,E2 13403.659} C_VEL
LIN {X 0,Y 417.091,Z 1182.034,A -85,B 0,C 180,E1 13400.896,E2 13400.896} C_VEL
LIN {X 0,Y 418.159,Z 1176.283,A -85,B 0,C 180,E1 13397.958,E2 13397.958} C_VEL
LIN {X 0,Y 419.637,Z 1169.605,A -85,B 0,C 180,E1 13395.088,E2 13395.088} C_VEL
LIN {X 0,Y 421.822,Z 1161.338,A -85,B 0,C 180,E1 13392.052,E2 13392.052} C_VEL
LIN {X 0,Y 425.569,Z 1148.868,A -85,B 0,C 180,E1 13388.209,E2 13388.209} C_VEL
LIN {X 0,Y 429.299,Z 1137.658,A -85,B 0,C 180,E1 13385.28,E2 13385.28} C_VEL
LIN {X 0,Y 433.291,Z 1126.269,A -85,B 0,C 180,E1 13382.663,E2 13382.663} C_VEL
LIN {X 0,Y 438.07,Z 1113.178,A -85,B 0,C 180,E1 13380.009,E2 13380.009} C_VEL
LIN {X 0,Y 444.769,Z 1095.345,A -85,B 0,C 180,E1 13376.887,E2 13376.887} C_VEL
LIN {X 0,Y 450.758,Z 1079.269,A -85,B 0,C 180,E1 13374.467,E2 13374.467} C_VEL
LIN {X 0,Y 456.286,Z 1064.282,A -85,B 0,C 180,E1 13372.469,E2 13372.469} C_VEL
LIN {X 0,Y 462.012,Z 1048.437,A -85,B 0,C 180,E1 13370.59,E2 13370.59} C_VEL
LIN {X 0,Y 468.482,Z 1029.951,A -85,B 0,C 180,E1 13368.657,E2 13368.657} C_VEL
LIN {X 0,Y 476.305,Z 1006.267,A -85,B 0,C 180,E1 13366.534,E2 13366.534} C_VEL
LIN {X 0,Y 482.116,Z 987.355,A -85,B 0,C 180,E1 13365.075,E2 13365.075} C_VEL
LIN {X 0,Y 487.545,Z 968.363,A -85,B 0,C 180,E1 13363.788,E2 13363.788} C_VEL
LIN {X 0,Y 492.683,Z 948.99,A -85,B 0,C 180,E1 13362.645,E2 13362.645} C_VEL
LIN {X 0,Y 497.792,Z 927.824,A -85,B 0,C 180,E1 13361.564,E2 13361.564} C_VEL
LIN {X 0,Y 503.692,Z 899.725,A -85,B 0,C 180,E1 13360.378,E2 13360.378} C_VEL
LIN {X 0,Y 507.691,Z 876.982,A -85,B 0,C 180,E1 13359.602,E2 13359.602} C_VEL
LIN {X 0,Y 510.835,Z 855.844,A -85,B 0,C 180,E1 13359.013,E2 13359.013} C_VEL
LIN {X 0,Y 513.476,Z 833.913,A -85,B 0,C 180,E1 13358.525,E2 13358.525} C_VEL
LIN {X 0,Y 515.806,Z 805.5,A -85,B 0,C 180,E1 13358.03,E2 13358.03} C_VEL
LIN {X 0,Y 528.448,Z 580.869,A -85,B 0,C 180,E1 13354.568,E2 13354.568} C_VEL
LIN {X 0,Y 533.229,Z 497.749,A -85,B 0,C 180,E1 13353.263,E2 13353.263} C_VEL
LIN {X 0,Y 522.522,Z 481.845,A -85,B 0,C 180,E1 13350.662,E2 13350.662} C_VEL
LIN {X 0,Y 512.314,Z 467.519,A -85,B 0,C 180,E1 13347.868,E2 13347.868} C_VEL
LIN {X 0,Y 503.747,Z 456.162,A -85,B 0,C 180,E1 13345.199,E2 13345.199} C_VEL
LIN {X 0,Y 499.509,Z 450.646,A -85,B 0,C 180,E1 13343.725,E2 13343.725} C_VEL
LIN {X 0,Y 495.977,Z 446.087,A -85,B 0,C 180,E1 13342.397,E2 13342.397} C_VEL
LIN {X 0,Y 491.873,Z 440.907,A -85,B 0,C 180,E1 13340.715,E2 13340.715} C_VEL
LIN {X 0,Y 488.151,Z 436.127,A -85,B 0,C 180,E1 13339.007,E2 13339.007} C_VEL
LIN {X 0,Y 484.119,Z 431.497,A -85,B 0,C 180,E1 13336.931,E2 13336.931} C_VEL
LIN {X 0,Y 482.937,Z 429.789,A -85,B 0,C 180,E1 13336.231,E2 13336.231} C_VEL
LIN {X 0,Y 479.456,Z 426.107,A -85,B 0,C 180,E1 13334,E2 13334} C_VEL
LIN {X 0,Y 478.134,Z 423.737,A -85,B 0,C 180,E1 13332.93,E2 13332.93} C_VEL
LIN {X 0,Y 474.765,Z 420.854,A -85,B 0,C 180,E1 13329.822,E2 13329.822} C_VEL
LIN {X 0,Y 473.322,Z 417.55,A -85,B 0,C 180,E1 13327.526,E2 13327.526} C_VEL
LIN {X 0,Y 472.162,Z 417.175,A -85,B 0,C 180,E1 13321.335,E2 13321.335} C_VEL
LIN {X 0,Y 473.468,Z 417.811,A -85,B 0,C 180,E1 13318.306,E2 13318.306} C_VEL
LIN {X 0,Y 475.193,Z 421.512,A -85,B 0,C 180,E1 13315.777,E2 13315.777} C_VEL
LIN {X 0,Y 478.449,Z 424.189,A -85,B 0,C 180,E1 13312.917,E2 13312.917} C_VEL
LIN {X 0,Y 481.366,Z 428.565,A -85,B 0,C 180,E1 13310.796,E2 13310.796} C_VEL
LIN {X 0,Y 483.449,Z 430.396,A -85,B 0,C 180,E1 13309.574,E2 13309.574} C_VEL
LIN {X 0,Y 486.605,Z 434.611,A -85,B 0,C 180,E1 13307.841,E2 13307.841} C_VEL
LIN {X 0,Y 488.257,Z 436.328,A -85,B 0,C 180,E1 13307.042,E2 13307.042} C_VEL
LIN {X 0,Y 491.973,Z 441.107,A -85,B 0,C 180,E1 13305.343,E2 13305.343} C_VEL
LIN {X 0,Y 497.65,Z 448.309,A -85,B 0,C 180,E1 13303.062,E2 13303.062} C_VEL
LIN {X 0,Y 502.28,Z 454.375,A -85,B 0,C 180,E1 13301.397,E2 13301.397} C_VEL
LIN {X 0,Y 508.816,Z 462.783,A -85,B 0,C 180,E1 13299.285,E2 13299.285} C_VEL
LIN {X 0,Y 515.636,Z 472.594,A -85,B 0,C 180,E1 13297.271,E2 13297.271} C_VEL
LIN {X 0,Y 526.359,Z 489.249,A -85,B 0,C 180,E1 13294.425,E2 13294.425} C_VEL
LIN {X 0,Y 533.26,Z 500.836,A -85,B 0,C 180,E1 13292.753,E2 13292.753} C_VEL
LIN {X 0,Y 520.908,Z 715.717,A -85,B 0,C 180,E1 13289.432,E2 13289.432} C_VEL
LIN {X 0,Y 514.641,Z 825.591,A -85,B 0,C 180,E1 13287.724,E2 13287.724} C_VEL
LIN {X 0,Y 511.89,Z 853.081,A -85,B 0,C 180,E1 13287.197,E2 13287.197} C_VEL
LIN {X 0,Y 508.079,Z 879.413,A -85,B 0,C 180,E1 13286.511,E2 13286.511} C_VEL
LIN {X 0,Y 504.348,Z 900.922,A -85,B 0,C 180,E1 13285.813,E2 13285.813} C_VEL
LIN {X 0,Y 500.314,Z 921.213,A -85,B 0,C 180,E1 13285.024,E2 13285.024} C_VEL
LIN {X 0,Y 495.434,Z 942.96,A -85,B 0,C 180,E1 13284.027,E2 13284.027} C_VEL
LIN {X 0,Y 488.664,Z 969.728,A -85,B 0,C 180,E1 13282.552,E2 13282.552} C_VEL
LIN {X 0,Y 482.893,Z 990.132,A -85,B 0,C 180,E1 13281.223,E2 13281.223} C_VEL
LIN {X 0,Y 477.352,Z 1008.374,A -85,B 0,C 180,E1 13279.867,E2 13279.867} C_VEL
LIN {X 0,Y 471.39,Z 1026.896,A -85,B 0,C 180,E1 13278.3,E2 13278.3} C_VEL
LIN {X 0,Y 464.672,Z 1046.865,A -85,B 0,C 180,E1 13276.371,E2 13276.371} C_VEL
LIN {X 0,Y 457.159,Z 1068.068,A -85,B 0,C 180,E1 13273.98,E2 13273.98} C_VEL
LIN {X 0,Y 451.158,Z 1084.531,A -85,B 0,C 180,E1 13271.843,E2 13271.843} C_VEL
LIN {X 0,Y 445.774,Z 1099.156,A -85,B 0,C 180,E1 13269.703,E2 13269.703} C_VEL
LIN {X 0,Y 440.441,Z 1113.657,A -85,B 0,C 180,E1 13267.311,E2 13267.311} C_VEL
LIN {X 0,Y 434.433,Z 1130.303,A -85,B 0,C 180,E1 13264.166,E2 13264.166} C_VEL
LIN {X 0,Y 429.615,Z 1144.073,A -85,B 0,C 180,E1 13261.11,E2 13261.11} C_VEL
LIN {X 0,Y 425.98,Z 1155.151,A -85,B 0,C 180,E1 13258.304,E2 13258.304} C_VEL
LIN {X 0,Y 422.994,Z 1165.04,A -85,B 0,C 180,E1 13255.446,E2 13255.446} C_VEL
LIN {X 0,Y 420.115,Z 1175.892,A -85,B 0,C 180,E1 13251.795,E2 13251.795} C_VEL
LIN {X 0,Y 418.2,Z 1184.279,A -85,B 0,C 180,E1 13248.34,E2 13248.34} C_VEL
LIN {X 0,Y 417.15,Z 1190.195,A -85,B 0,C 180,E1 13245.43,E2 13245.43} C_VEL
LIN {X 0,Y 416.489,Z 1194.918,A -85,B 0,C 180,E1 13242.619,E2 13242.619} C_VEL
LIN {X 0,Y 416.138,Z 1198.67,A -85,B 0,C 180,E1 13239.823,E2 13239.823} C_VEL
LIN {X 0,Y 415.973,Z 1201.474,A -85,B 0,C 180,E1 13237.042,E2 13237.042} C_VEL
LIN {X 0,Y 415.917,Z 1203.35,A -85,B 0,C 180,E1 13234.274,E2 13234.274} C_VEL
LIN {X 0,Y 415.911,Z 1204.308,A -85,B 0,C 180,E1 13231.516,E2 13231.516} C_VEL
LIN {X 0,Y 415.912,Z 1204.375,A -85,B 0,C 180,E1 13228.899,E2 13228.899} C_VEL
LIN {X 0,Y 415.915,Z 1203.536,A -85,B 0,C 180,E1 13226.11,E2 13226.11} C_VEL
LIN {X 0,Y 415.961,Z 1201.81,A -85,B 0,C 180,E1 13223.375,E2 13223.375} C_VEL
LIN {X 0,Y 416.101,Z 1199.141,A -85,B 0,C 180,E1 13220.596,E2 13220.596} C_VEL
LIN {X 0,Y 416.444,Z 1195.32,A -85,B 0,C 180,E1 13217.662,E2 13217.662} C_VEL
LIN {X 0,Y 417.066,Z 1190.696,A -85,B 0,C 180,E1 13214.852,E2 13214.852} C_VEL
LIN {X 0,Y 418.103,Z 1184.777,A -85,B 0,C 180,E1 13211.888,E2 13211.888} C_VEL
LIN {X 0,Y 419.752,Z 1177.385,A -85,B 0,C 180,E1 13208.773,E2 13208.773} C_VEL
LIN {X 0,Y 422.662,Z 1166.549,A -85,B 0,C 180,E1 13204.948,E2 13204.948} C_VEL
LIN {X 0,Y 426.028,Z 1155.578,A -85,B 0,C 180,E1 13201.701,E2 13201.701} C_VEL
LIN {X 0,Y 429.703,Z 1144.749,A -85,B 0,C 180,E1 13198.898,E2 13198.898} C_VEL
LIN {X 0,Y 434.082,Z 1132.593,A -85,B 0,C 180,E1 13196.123,E2 13196.123} C_VEL
LIN {X 0,Y 440.464,Z 1115.938,A -85,B 0,C 180,E1 13192.826,E2 13192.826} C_VEL
LIN {X 0,Y 446.498,Z 1100.345,A -85,B 0,C 180,E1 13190.175,E2 13190.175} C_VEL
LIN {X 0,Y 452.301,Z 1085.511,A -85,B 0,C 180,E1 13187.947,E2 13187.947} C_VEL
LIN {X 0,Y 458.411,Z 1069.821,A -85,B 0,C 180,E1 13185.858,E2 13185.858} C_VEL
LIN {X 0,Y 465.351,Z 1051.69,A -85,B 0,C 180,E1 13183.733,E2 13183.733} C_VEL
LIN {X 0,Y 473.614,Z 1029.061,A -85,B 0,C 180,E1 13181.457,E2 13181.457} C_VEL
LIN {X 0,Y 480.254,Z 1009.922,A -85,B 0,C 180,E1 13179.804,E2 13179.804} C_VEL
LIN {X 0,Y 486.253,Z 991.686,A -85,B 0,C 180,E1 13178.424,E2 13178.424} C_VEL
LIN {X 0,Y 491.704,Z 973.952,A -85,B 0,C 180,E1 13177.241,E2 13177.241} C_VEL
LIN {X 0,Y 497.339,Z 954.102,A -85,B 0,C 180,E1 13176.081,E2 13176.081} C_VEL
LIN {X 0,Y 503.778,Z 929.265,A -85,B 0,C 180,E1 13174.847,E2 13174.847} C_VEL
LIN {X 0,Y 509.372,Z 903.726,A -85,B 0,C 180,E1 13173.818,E2 13173.818} C_VEL
LIN {X 0,Y 513.449,Z 882.367,A -85,B 0,C 180,E1 13173.112,E2 13173.112} C_VEL
LIN {X 0,Y 516.843,Z 861.258,A -85,B 0,C 180,E1 13172.538,E2 13172.538} C_VEL
LIN {X 0,Y 519.884,Z 837.935,A -85,B 0,C 180,E1 13172.039,E2 13172.039} C_VEL
LIN {X 0,Y 522.769,Z 802.028,A -85,B 0,C 180,E1 13171.434,E2 13171.434} C_VEL
LIN {X 0,Y 536.924,Z 580.641,A -85,B 0,C 180,E1 13167.988,E2 13167.988} C_VEL
LIN {X 0,Y 542.029,Z 503.874,A -85,B 0,C 180,E1 13166.781,E2 13166.781} C_VEL
LIN {X 0,Y 535.465,Z 493.172,A -85,B 0,C 180,E1 13164.815,E2 13164.815} C_VEL
LIN {X 0,Y 527.324,Z 480.46,A -85,B 0,C 180,E1 13162.052,E2 13162.052} C_VEL
LIN {X 0,Y 521.729,Z 472.701,A -85,B 0,C 180,E1 13159.888,E2 13159.888} C_VEL
LIN {X 0,Y 517.803,Z 467.501,A -85,B 0,C 180,E1 13158.171,E2 13158.171} C_VEL
LIN {X 0,Y 514.198,Z 462.63,A -85,B 0,C 180,E1 13156.377,E2 13156.377} C_VEL
LIN {X 0,Y 510.595,Z 457.869,A -85,B 0,C 180,E1 13154.285,E2 13154.285} C_VEL
LIN {X 0,Y 506.858,Z 453.456,A -85,B 0,C 180,E1 13151.608,E2 13151.608} C_VEL
LIN {X 0,Y 505.787,Z 451.505,A -85,B 0,C 180,E1 13150.594,E2 13150.594} C_VEL
LIN {X 0,Y 502.523,Z 448.15,A -85,B 0,C 180,E1 13146.398,E2 13146.398} C_VEL
LIN {X 0,Y 501.911,Z 445.492,A -85,B 0,C 180,E1 13143.426,E2 13143.426} C_VEL
LIN {X 0,Y 501.934,Z 445.73,A -85,B 0,C 180,E1 13141.941,E2 13141.941} C_VEL
LIN {X 0,Y 504.799,Z 450.868,A -85,B 0,C 180,E1 13136.138,E2 13136.138} C_VEL
LIN {X 0,Y 506.107,Z 451.925,A -85,B 0,C 180,E1 13134.899,E2 13134.899} C_VEL
LIN {X 0,Y 508.664,Z 455.934,A -85,B 0,C 180,E1 13132.773,E2 13132.773} C_VEL
LIN {X 0,Y 510.613,Z 457.908,A -85,B 0,C 180,E1 13131.498,E2 13131.498} C_VEL
LIN {X 0,Y 513.894,Z 462.33,A -85,B 0,C 180,E1 13129.575,E2 13129.575} C_VEL
LIN {X 0,Y 515.257,Z 464.013,A -85,B 0,C 180,E1 13128.867,E2 13128.867} C_VEL
LIN {X 0,Y 519.356,Z 469.444,A -85,B 0,C 180,E1 13126.925,E2 13126.925} C_VEL
LIN {X 0,Y 523.957,Z 475.692,A -85,B 0,C 180,E1 13125.014,E2 13125.014} C_VEL
LIN {X 0,Y 529.597,Z 483.244,A -85,B 0,C 180,E1 13122.955,E2 13122.955} C_VEL
LIN {X 0,Y 537.832,Z 495.229,A -85,B 0,C 180,E1 13120.308,E2 13120.308} C_VEL
LIN {X 0,Y 542.081,Z 501.657,A -85,B 0,C 180,E1 13119.073,E2 13119.073} C_VEL
LIN {X 0,Y 528.314,Z 710.872,A -85,B 0,C 180,E1 13115.813,E2 13115.813} C_VEL
LIN {X 0,Y 521.27,Z 819.786,A -85,B 0,C 180,E1 13114.102,E2 13114.102} C_VEL
LIN {X 0,Y 518.291,Z 847.271,A -85,B 0,C 180,E1 13113.571,E2 13113.571} C_VEL
LIN {X 0,Y 514.283,Z 873.221,A -85,B 0,C 180,E1 13112.89,E2 13112.89} C_VEL
LIN {X 0,Y 510.387,Z 894.218,A -85,B 0,C 180,E1 13112.208,E2 13112.208} C_VEL
LIN {X 0,Y 506.101,Z 914.364,A -85,B 0,C 180,E1 13111.422,E2 13111.422} C_VEL
LIN {X 0,Y 501.324,Z 934.238,A -85,B 0,C 180,E1 13110.514,E2 13110.514} C_VEL
LIN {X 0,Y 495.611,Z 955.724,A -85,B 0,C 180,E1 13109.366,E2 13109.366} C_VEL
LIN {X 0,Y 488.133,Z 980.818,A -85,B 0,C 180,E1 13107.775,E2 13107.775} C_VEL
LIN {X 0,Y 481.516,Z 1001.032,A -85,B 0,C 180,E1 13106.267,E2 13106.267} C_VEL
LIN {X 0,Y 475.227,Z 1019.148,A -85,B 0,C 180,E1 13104.72,E2 13104.72} C_VEL
LIN {X 0,Y 468.576,Z 1037.401,A -85,B 0,C 180,E1 13102.944,E2 13102.944} C_VEL
LIN {X 0,Y 460.411,Z 1058.929,A -85,B 0,C 180,E1 13100.52,E2 13100.52} C_VEL
LIN {X 0,Y 453.417,Z 1076.62,A -85,B 0,C 180,E1 13098.189,E2 13098.189} C_VEL
LIN {X 0,Y 447.561,Z 1091.339,A -85,B 0,C 180,E1 13095.988,E2 13095.988} C_VEL
LIN {X 0,Y 442.003,Z 1105.354,A -85,B 0,C 180,E1 13093.622,E2 13093.622} C_VEL
LIN {X 0,Y 435.918,Z 1121.09,A -85,B 0,C 180,E1 13090.603,E2 13090.603} C_VEL
LIN {X 0,Y 430.425,Z 1135.594,A -85,B 0,C 180,E1 13087.322,E2 13087.322} C_VEL
LIN {X 0,Y 426.66,Z 1146.298,A -85,B 0,C 180,E1 13084.549,E2 13084.549} C_VEL
LIN {X 0,Y 423.589,Z 1155.768,A -85,B 0,C 180,E1 13081.761,E2 13081.761} C_VEL
LIN {X 0,Y 420.927,Z 1164.912,A -85,B 0,C 180,E1 13078.674,E2 13078.674} C_VEL
LIN {X 0,Y 418.501,Z 1174.732,A -85,B 0,C 180,E1 13074.714,E2 13074.714} C_VEL
LIN {X 0,Y 417.257,Z 1181.182,A -85,B 0,C 180,E1 13071.508,E2 13071.508} C_VEL
LIN {X 0,Y 416.531,Z 1186.101,A -85,B 0,C 180,E1 13068.52,E2 13068.52} C_VEL
LIN {X 0,Y 416.17,Z 1189.724,A -85,B 0,C 180,E1 13065.752,E2 13065.752} C_VEL
LIN {X 0,Y 415.983,Z 1192.504,A -85,B 0,C 180,E1 13062.916,E2 13062.916} C_VEL
LIN {X 0,Y 415.924,Z 1194.265,A -85,B 0,C 180,E1 13060.247,E2 13060.247} C_VEL
LIN {X 0,Y 415.919,Z 1194.564,A -85,B 0,C 180,E1 13059.633,E2 13059.633} C_VEL
LIN {X 0,Y 414.927,Z 1195.044,A -85,B 0,C 180,E1 13058.574,E2 13058.574} C_VEL
LIN {X 0,Y 408.437,Z 1195.485,A -85,B 0,C 180,E1 13055.584,E2 13055.584} C_VEL
LIN {X 0,Y 407.905,Z 1195.359,A -85,B 0,C 180,E1 13054.803,E2 13054.803} C_VEL
LIN {X 0,Y 407.925,Z 1194.533,A -85,B 0,C 180,E1 13051.966,E2 13051.966} C_VEL
LIN {X 0,Y 407.983,Z 1192.822,A -85,B 0,C 180,E1 13049.157,E2 13049.157} C_VEL
LIN {X 0,Y 408.148,Z 1190.224,A -85,B 0,C 180,E1 13046.348,E2 13046.348} C_VEL
LIN {X 0,Y 408.538,Z 1186.525,A -85,B 0,C 180,E1 13043.394,E2 13043.394} C_VEL
LIN {X 0,Y 409.196,Z 1182.065,A -85,B 0,C 180,E1 13040.577,E2 13040.577} C_VEL
LIN {X 0,Y 410.319,Z 1176.367,A -85,B 0,C 180,E1 13037.617,E2 13037.617} C_VEL
LIN {X 0,Y 411.917,Z 1169.596,A -85,B 0,C 180,E1 13034.657,E2 13034.657} C_VEL
LIN {X 0,Y 414.48,Z 1160.517,A -85,B 0,C 180,E1 13031.286,E2 13031.286} C_VEL
LIN {X 0,Y 418.202,Z 1148.789,A -85,B 0,C 180,E1 13027.656,E2 13027.656} C_VEL
LIN {X 0,Y 422.013,Z 1137.853,A -85,B 0,C 180,E1 13024.756,E2 13024.756} C_VEL
LIN {X 0,Y 426.075,Z 1126.748,A -85,B 0,C 180,E1 13022.16,E2 13022.16} C_VEL
LIN {X 0,Y 430.779,Z 1114.367,A -85,B 0,C 180,E1 13019.602,E2 13019.602} C_VEL
LIN {X 0,Y 437.078,Z 1098.335,A -85,B 0,C 180,E1 13016.699,E2 13016.699} C_VEL
LIN {X 0,Y 443.919,Z 1080.605,A -85,B 0,C 180,E1 13013.961,E2 13013.961} C_VEL
LIN {X 0,Y 449.908,Z 1064.944,A -85,B 0,C 180,E1 13011.842,E2 13011.842} C_VEL
LIN {X 0,Y 455.747,Z 1049.326,A -85,B 0,C 180,E1 13009.969,E2 13009.969} C_VEL
LIN {X 0,Y 461.833,Z 1032.481,A -85,B 0,C 180,E1 13008.177,E2 13008.177} C_VEL
LIN {X 0,Y 469.317,Z 1010.967,A -85,B 0,C 180,E1 13006.178,E2 13006.178} C_VEL
LIN {X 0,Y 476.508,Z 988.304,A -85,B 0,C 180,E1 13004.399,E2 13004.399} C_VEL
LIN {X 0,Y 482.083,Z 969.403,A -85,B 0,C 180,E1 13003.107,E2 13003.107} C_VEL
LIN {X 0,Y 487.378,Z 950.016,A -85,B 0,C 180,E1 13001.954,E2 13001.954} C_VEL
LIN {X 0,Y 492.318,Z 930.173,A -85,B 0,C 180,E1 13000.929,E2 13000.929} C_VEL
LIN {X 0,Y 497.973,Z 904.833,A -85,B 0,C 180,E1 12999.821,E2 12999.821} C_VEL
LIN {X 0,Y 502.798,Z 878.418,A -85,B 0,C 180,E1 12998.9,E2 12998.9} C_VEL
LIN {X 0,Y 506.085,Z 857.027,A -85,B 0,C 180,E1 12998.298,E2 12998.298} C_VEL
LIN {X 0,Y 508.759,Z 835.577,A -85,B 0,C 180,E1 12997.815,E2 12997.815} C_VEL
LIN {X 0,Y 510.922,Z 811.323,A -85,B 0,C 180,E1 12997.382,E2 12997.382} C_VEL
LIN {X 0,Y 523.917,Z 588.383,A -85,B 0,C 180,E1 12993.931,E2 12993.931} C_VEL
LIN {X 0,Y 529.075,Z 502.403,A -85,B 0,C 180,E1 12992.59,E2 12992.59} C_VEL
LIN {X 0,Y 519.09,Z 487.56,A -85,B 0,C 180,E1 12990.086,E2 12990.086} C_VEL
LIN {X 0,Y 509.913,Z 474.47,A -85,B 0,C 180,E1 12987.503,E2 12987.503} C_VEL
LIN {X 0,Y 501.816,Z 463.543,A -85,B 0,C 180,E1 12984.925,E2 12984.925} C_VEL
LIN {X 0,Y 497.337,Z 457.657,A -85,B 0,C 180,E1 12983.333,E2 12983.333} C_VEL
LIN {X 0,Y 494.016,Z 453.336,A -85,B 0,C 180,E1 12982.052,E2 12982.052} C_VEL
LIN {X 0,Y 490.126,Z 448.347,A -85,B 0,C 180,E1 12980.417,E2 12980.417} C_VEL
LIN {X 0,Y 485.887,Z 442.972,A -85,B 0,C 180,E1 12978.414,E2 12978.414} C_VEL
LIN {X 0,Y 482.45,Z 438.726,A -85,B 0,C 180,E1 12976.557,E2 12976.557} C_VEL
LIN {X 0,Y 481.576,Z 437.531,A -85,B 0,C 180,E1 12976.03,E2 12976.03} C_VEL
LIN {X 0,Y 478.164,Z 433.808,A -85,B 0,C 180,E1 12973.791,E2 12973.791} C_VEL
LIN {X 0,Y 477.019,Z 431.627,A -85,B 0,C 180,E1 12972.838,E2 12972.838} C_VEL
LIN {X 0,Y 473.692,Z 428.743,A -85,B 0,C 180,E1 12969.722,E2 12969.722} C_VEL
LIN {X 0,Y 472.279,Z 425.477,A -85,B 0,C 180,E1 12967.42,E2 12967.42} C_VEL
LIN {X 0,Y 471.184,Z 425.115,A -85,B 0,C 180,E1 12961.338,E2 12961.338} C_VEL
LIN {X 0,Y 472.416,Z 425.709,A -85,B 0,C 180,E1 12958.423,E2 12958.423} C_VEL
LIN {X 0,Y 474.212,Z 429.51,A -85,B 0,C 180,E1 12955.768,E2 12955.768} C_VEL
LIN {X 0,Y 477.302,Z 432.173,A -85,B 0,C 180,E1 12953.021,E2 12953.021} C_VEL
LIN {X 0,Y 480.2,Z 436.446,A -85,B 0,C 180,E1 12950.895,E2 12950.895} C_VEL
LIN {X 0,Y 482.153,Z 438.269,A -85,B 0,C 180,E1 12949.726,E2 12949.726} C_VEL
LIN {X 0,Y 485.512,Z 442.619,A -85,B 0,C 180,E1 12947.874,E2 12947.874} C_VEL
LIN {X 0,Y 486.901,Z 444.244,A -85,B 0,C 180,E1 12947.186,E2 12947.186} C_VEL
LIN {X 0,Y 490.596,Z 448.908,A -85,B 0,C 180,E1 12945.482,E2 12945.482} C_VEL
LIN {X 0,Y 496.136,Z 456.174,A -85,B 0,C 180,E1 12943.22,E2 12943.22} C_VEL
